// SIMATIC STEP 7 (V5.x) project e009v440
// CPU: CPU 313C-2 DP
// station: P_ADR_BUS
// station: Hardware
// station: PLC Roll Forming
// program: Programa S7(8)
// program: CU320
// program: CU320-2 DP
// program: M440
// program: M440
// program: M440

SYMBOL_TABLE
"Tendencia"	DB 1	DB 1
"EncóderPerfilador"	DB 2	DB 2
"Datos Pieza - Receta"	DB 3	DB 3
"Datos Pieza - Alm1"	DB 4	DB 4
"Datos Pieza - Alm2"	DB 5	DB 5
"Datos Pieza - Araña"	DB 6	DB 6
"Datos Pieza - Rolos"	DB 7	DB 7
"Datos Pieza - Perfilador"	DB 8	DB 8
"Datos Pieza - Cinta"	DB 9	DB 9
"Datos Pieza - Pinza"	DB 10	DB 10
"Datos Pieza - Plegadores"	DB 11	DB 11
"Datos Pieza - Descargado"	DB 12	DB 12
"Posiciones_Pinza"	DB 13	DB 13
"Datos Pieza - VACIO"	DB 14	DB 14
"Ultimo Estado"	DB 15	DB 15
"Datos Cosntructivos"	DB 16	DB 16
"Posiciones Pinza 00"	DB 17	DB 17
"Posiciones_Pinza_Ant"	DB 18	DB 18
"DB Asistencia"	DB 19	DB 19
"ReglasBalluff"	DB 20	DB 20
"Referenciado"	DB 21	DB 21
"Posiciones_Pinza_Ant2"	DB 23	DB 23
"Posiciones_Pinza_Ant3"	DB 24	DB 24
"PosReal_Pinza"	DB 25	DB 25
"PosReal_Pinza_Ant"	DB 26	DB 26
"PosReal_Pinza_Ant2"	DB 27	DB 27
"PosReal_Pinza_Ant3"	DB 28	DB 28
"Error_Pinza_Ant"	DB 29	DB 29
"DB_OP"	DB 50	DB 50
"Recetas"	DB 51	DB 51
"OFFSET"	DB 52	DB 52
"Posiciones Pinza"	DB 53	DB 53
"Posiciones Plegador 2"	DB 54	DB 54
"Posiciones Plegador 1"	DB 55	DB 55
"Posiciones Plegadores 00"	DB 56	DB 56
"Posiciones Pleg. 1 Ant"	DB 57	DB 57
"Posiciones Pleg. 2 Ant"	DB 58	DB 58
"Homing Plegadores"	FC 1	FC 1
"ModoMix"	FC 2	FC 2
"Manual Selección Mov."	FC 4	FC 4
"General"	FC 5	FC 5
"Generador de Fallas"	FC 6	FC 6
"Asistencia"	FC 8	FC 8
"Control de Plegadora"	FC 9	FC 9
"Perfilador"	FC 10	FC 10
"Transportes"	FC 11	FC 11
"Control de Pinza y Forma"	FC 12	FC 12
"Controlador Posiciones"	FC 13	FC 13
"Almacenes"	FC 15	FC 15
"Registro_pos_Plegador"	FC 17	FC 17
"Registro_pos_Pinza"	FC 18	FC 18
"Araña"	FC 20	FC 20
"Plegadora"	FC 30	FC 30
"Plegador 1"	FC 31	FC 31
"Descarga"	FC 40	FC 40
"TR_MP"	FC 50	FC 50
"Gestión de Datos"	FC 51	FC 51
"eProC - Máquina Estados"	FC 150	FC 150
"23S1"	I 0.0	BOOL	// Pupitre Almacenes - Rearme
"23SH2"	I 0.1	BOOL	// Pupitre Almacenes - Reconocimiento
"Pair"	I 0.2	BOOL	// Presión de Aire
"GH_Tmax"	I 0.3	BOOL	// Grupo áulico (23S8) - Temperatura máxima
"23S3"	I 0.4	BOOL	// Pupitre Principal : Rearme
"23S5"	I 0.5	BOOL	// Alineador Eje Y Plegador 1 ON
"23S6"	I 0.6	BOOL	// Alineador Eje Y Plegador 1 OFF
"23S4"	I 0.7	BOOL	// Presostato Freno Perfilador
"24S1_01"	I 1.0	BOOL	// Rueda Unidades :1
"24S1_02"	I 1.1	BOOL	// Rueda Unidades :2
"24S1_04"	I 1.2	BOOL	// Rueda Unidades :4
"24S1_08"	I 1.3	BOOL	// Rueda Unidades :8
"24S1_10"	I 1.4	BOOL	// Rueda Decenas :1
"24S1_20"	I 1.5	BOOL	// Rueda Decenas :2
"24S1_40"	I 1.6	BOOL	// Rueda Decenas :4
"24S1_80"	I 1.7	BOOL	// Rueda Decenas :8
"QF9"	I 2.0	BOOL	// Térmico Freno Ajuste de Formado
"25S2"	I 2.1	BOOL	// Desaceleración Transporte Cinta
"25S3"	I 2.2	BOOL	// Fin de Carrera Araña Arriba
"25S4"	I 2.3	BOOL	// Pistón 1 Araña Contraído
"25S5"	I 2.4	BOOL	// Fin de Carrera Araña Abajo
"25S6"	I 2.5	BOOL	// Araña Abajo
"25S7"	I 2.6	BOOL	// Pistón 2 Araña Expandido
"25S8"	I 2.7	BOOL	// Pistón 2 Araña Contraído
"26S1"	I 3.0	BOOL	// Tulipas no apoyadas en Chapa
"26S2"	I 3.1	BOOL	// Araña en Posicion de Carga
"26S3"	I 3.2	BOOL	// Araña en Posición de Descarga
"26S4"	I 3.3	BOOL	// Bajar Velocidad Transporte de Araña para Tomar Chapa
"26S5"	I 3.4	BOOL	// Bajar Velocidad Transporte de Araña para Soltar Chapa
"26S6"	I 3.5	BOOL	// Presencia de Almacén 2 en Puesto de Espera
"26S7"	I 3.6	BOOL	// Presencia de Almacén 2 en Puesto de Trabajo
"26S8"	I 3.7	BOOL	// Presencia de Chapa en Transporte Rolos
"27S1"	I 4.0	BOOL	// Pulsador Avance Perfilador
"27S2"	I 4.1	BOOL	// Pulsador Retroceso Perfilador
"27S3"	I 4.2	BOOL	// Chapa en entrada Perfilador
"27S4"	I 4.3	BOOL	// Chapa en salida Perfilador
"27S5"	I 4.4	BOOL	// Formador Herramienta 1 Martillo Off
"27S6"	I 4.5	BOOL	// Formador Herramienta 1 Martillo On
"27S7"	I 4.6	BOOL	// Formador Herramienta 1 Matriz Off
"27S8"	I 4.7	BOOL	// Formador Herramienta 1 Matriz On
"28S1"	I 5.0	BOOL	// Formador Herramienta 2 Martillo Off
"28S2"	I 5.1	BOOL	// Formador Herramienta 2 Martillo On
"28S3"	I 5.2	BOOL	// Formador Herramienta 2 Matriz Off
"28S4"	I 5.3	BOOL	// Formador Herramienta 2 Matriz On
"28S5"	I 5.4	BOOL	// Formador Bloqueo Herramienta On
"28S6"	I 5.5	BOOL	// Matriz Formadora Bloqueo Herramienta Off
"28S7"	I 5.6	BOOL	// Ajuste Formador Fin de Carrera Mín.
"28S8"	I 5.7	BOOL	// Ajuste Formador Fin de Carrera Máx.
"29S1"	I 6.0	BOOL	// Formador Bloqueo de avance On
"29S2"	I 6.1	BOOL	// Formador Bloqueo de avance Off
"29S3"	I 6.2	BOOL	// Presencia de Chapa en Formador
"29S4"	I 6.3	BOOL	// Pinza Abierta
"29S5"	I 6.4	BOOL	// Pinza Cerrada
"29S6"	I 6.5	BOOL	// Ajuste Ancho Perfilador Fin de carrera Mín.
"29S7"	I 6.6	BOOL	// Ajuste Ancho Perfilador Fin de carrera Máx.
"29S8"	I 6.7	BOOL	// Plegadora Termostato Grupo Hidráulico
"30S1"	I 7.0	BOOL	// Plegadora Tenaza adelante
"30S2"	I 7.1	BOOL	// Plegadora Tenaza atrás
"30S3"	I 7.2	BOOL	// Plegadora Tenaza arriba
"30S4"	I 7.3	BOOL	// Plegadora Tenaza abajo
"30S5"	I 7.4	BOOL	// Plegadora Tenaza abierta
"30S6"	I 7.5	BOOL	// Plegadora Tenaza cerrada
"30S7"	I 7.6	BOOL	// Plegador 1 Cepillos Arriba
"30S8"	I 7.7	BOOL	// Plegador 1 Cepillos Abajo
"31S1"	I 8.0	BOOL	// Presencia de Producto en Descargador
"31S2"	I 8.1	BOOL	// Descargador Adelante
"31S3"	I 8.2	BOOL	// Descargador Atrás
"31S4"	I 8.3	BOOL	// Barrera Seguridad Descargador
"31S5"	I 8.4	BOOL	// Plegador 1 Fijación Arriba
"31S6"	I 8.5	BOOL	// Plegador 1 Fijación Abajo
"31S7"	I 8.6	BOOL	// Plegador 1 Arriba
"31S8"	I 8.7	BOOL	// Pieza en Descargador
"32S1"	I 9.0	BOOL	// Plegador 1 Prensa Abajo
"32S2"	I 9.1	BOOL	// Plegador 1 Prensa Arriba
"32S3"	I 9.2	BOOL	// Plegador 1 Extensión 1 Prensa Abajo
"32S4"	I 9.3	BOOL	// Plegador 1 Extensión 1 Prensa Arriba
"32S5"	I 9.4	BOOL	// Plegador 1 Extensión 2 Prensa Abajo
"32S6"	I 9.5	BOOL	// Plegador 1 Extensión 2 Prensa Arriba
"QM13.2"	I 9.6	BOOL	// Térmico Refrigeración Grupo Hidráulico Plegadora
"QM14"	I 9.7	BOOL	// Térmico Calentador de Chapa
"QM01"	I 10.0	BOOL	// Térmico Intercambiador de Almacenes
"VAR02"	I 10.1	BOOL	// Defecto Variador Araña
"VAR03"	I 10.2	BOOL	// Defecto Variador Transporte Rolos
"Reserva"	I 10.3	BOOL	// Reserva
"Reserva2"	I 10.4	BOOL	// Reserva
"Doble_Chapa_Perf"	I 10.5	BOOL	// Doble Espesor de Chapa en entrada de Perfilador
"Reserva3"	I 10.6	BOOL	// Reserva
"QM05"	I 10.7	BOOL	// Térmico Bombas de Lubricación Perfilador
"QM06"	I 11.0	BOOL	// Térmico Grupo Hidráulico Freno Perfilador
"QM07"	I 11.1	BOOL	// Térmico Ajuste de Ancho Perfilador
"VAR08"	I 11.2	BOOL	// Defecto Variador Transporte Cinta
"QM09"	I 11.3	BOOL	// Térmico Ajuste de Formado
"Sinamics_OK"	I 11.4	BOOL	// Smart Line Plegador Listo
"Sinamics_Alarme"	I 11.5	BOOL	// Defecto SmartLine Plegadora
"Carter"	I 11.6	BOOL	// Cubierta Perfilador abierta
"QM13.1"	I 11.7	BOOL	// Térmico Grupo Hidráulico Plegadora
"35S1"	I 12.0	BOOL	// Plegador 2 Fijación Arriba
"35S2"	I 12.1	BOOL	// Plegador 2 Fijación Abajo
"35S3"	I 12.2	BOOL	// Plegador 2 Arriba
"35S4"	I 12.3	BOOL	// Plegador 2 Abajo
"35S5"	I 12.4	BOOL	// Plegador 2 Prensa Abajo
"35S6"	I 12.5	BOOL	// Plegador 2 Prensa Arriba
"35S7"	I 12.6	BOOL	// Plegador 2 Extensión 1 Prensa Abajo
"35S8"	I 12.7	BOOL	// Plegador 2 Extensión 1 Prensa Arriba
"36S7"	I 13.0	BOOL	// Plegador 2 Extensión 2 Prensa Abajo
"36S8"	I 13.1	BOOL	// Plegador 2 Extensión 2 Prensa Arriba
"36S1"	I 13.2	BOOL	// Alineador Eje X Plegador 2 ON
"36S2"	I 13.3	BOOL	// Alineador Eje X Plegador 2 OFF
"36S3"	I 13.4	BOOL	// Alineador Eje Y Plegador 2 ON
"36S4"	I 13.5	BOOL	// Alineador Eje Y Plegador 2 OFF
"36S5"	I 13.6	BOOL	// Plegador 2 Cepillos Arriba
"36S6"	I 13.7	BOOL	// Plegador 2 Cepillos Abajo
"36S9"	I 14.0	BOOL	// Plegador 1 Prensa en Posición Intermedia
"36S17"	I 14.1	BOOL	// Plegador 2 Prensa en Posición Intermedia
"36S11"	I 14.2	BOOL	// Pinza Plegadora en Posición Intermedia
"36S12"	I 14.3	BOOL	// Descargador en Posición Intermedia
"36S13"	I 14.4	BOOL	// Atasco Perfilador Sensor 1
"36S14"	I 14.5	BOOL	// Atasco Perfilador Sensor 2
"36S15"	I 14.6	BOOL	// Atasco Perfilador Sensor 3
"36S16"	I 14.7	BOOL	// Atasco Perfilador Sensor 4
"36S10"	I 15.0	BOOL	// Barrera Almacenes
"36S18"	I 15.1	BOOL
"Reserva4"	I 15.2	BOOL	// Reserva
"iPLs_HabAlmacenes"	I 15.3	BOOL	// Pulsador Habilitación Almacenes
"iSel_Homming"	I 15.4	BOOL	// Selectora Habilitación Referenciado Plegadores
"31S7b"	I 15.5	BOOL	// Plegador 1 posición Arriba (pata)
"35S3b"	I 15.6	BOOL	// Plegador 2 posición Arriba (pata)
"36S70"	I 15.7	BOOL	// Barrera Atasco en Perfilador
"Atasco_6"	I 16.0	BOOL	// Sensor 6 Atasco Perfilador
"Atasco_7"	I 16.1	BOOL	// Sensor 7 Atasco Perfilador
"Atasco_8"	I 16.2	BOOL	// Sensor 8 Atasco Perfilador
"Atasco_9"	I 16.3	BOOL	// Sensor 9 Atasco Perfilador
"Atasco_10"	I 16.4	BOOL	// Sensor 10 Atasco Perfilador
"Atasco_11"	I 16.5	BOOL	// Sensor 11 Atasco Perfilador
"Atasco_12"	I 16.6	BOOL	// Sensor 12 Atasco Perfilador
"Atasco_13"	I 16.7	BOOL	// Sensor 13 Atasco Perfilador
"Atasco_14"	I 17.0	BOOL	// Sensor 14 Atasco Perfilador
"Atasco_15"	I 17.1	BOOL	// Sensor 15 Atasco Perfilador
"Atasco_16"	I 17.2	BOOL	// Sensor 16 Atasco Perfilador
"Atasco_17"	I 17.3	BOOL	// Sensor 17 Atasco Perfilador
"Atasco_18"	I 17.4	BOOL	// Sensor 18 Atasco Perfilador
"Atasco_19"	I 17.5	BOOL	// Sensor 19 Atasco Perfilador
"Atasco_21"	I 17.6	BOOL	// Sensor 21 Atasco Perfilador
"iSns_Perf_Atasco_16"	I 17.7	BOOL	// Sensor 20 Atasco Perfilador
"Atasco_22"	I 18.0	BOOL	// Sensor 22 Atasco Perfilador
"Atasco_23"	I 18.1	BOOL	// Sensor 23 Atasco Perfilador
"Atasco_24"	I 18.2	BOOL	// Sensor 24 Atasco Perfilador
"Atasco_5"	I 18.3	BOOL	// Sensor 5 Atasco Perfilador
"Safety_Barrera_Entrada"	I 19.0	BOOL	// Entrada desde PLC Safety en reemplazo de barrera de entrada original
"Safety_Corte_1"	I 19.1	BOOL	// Entrada desde PLC Safety para corte 1
"Safety_Corte_2"	I 19.2	BOOL	// Entrada desde PLC Safety para corte 2
"PRF_SLM_DATA0"	I 24.0	BOOL
"PRF_SLM_MS"	I 24.1	BOOL	// SmartLine Perfilador Mando Solicitado
"PRF_SLM_DATA01"	I 24.2	BOOL
"PRF_SLM_PREC"	I 24.3	BOOL	// SmartLine Perfilador Precarga Terminada
"PRF_SLM_CTC"	I 24.4	BOOL	// SmartLine Perfilador Contactor de Red Cerrado
"PRF_SLM_DATA02"	I 24.5	BOOL
"PRF_SLM_DATA03"	I 24.6	BOOL
"PRF_SLM_DATA04"	I 24.7	BOOL
"PRF_SLM_LC"	I 25.0	BOOL	// SmartLine Perfilador Listo Conexión
"PRF_SLM_LS"	I 25.1	BOOL	// SmartLine Perfilador Listo para Servicio
"PRF_SLM_SH"	I 25.2	BOOL	// SmartLine Perfilador Servicio Habilitado
"PRF_SLM_FA"	I 25.3	BOOL	// SmartLine Perfilador Fallo Activo  (0=NO, 1=SI)
"PRF_SLM_DES2A"	I 25.4	BOOL	// SmartLine Perfilador Sin Parada Natural Activa
"PRF_SLM_DES3A"	I 25.5	BOOL	// SmartLine Perfilador Sin Parada Rápida Activa
"PRF_SLM_BC"	I 25.6	BOOL	// SmartLine Perfilador Bloqueo de Conexión Activo
"PRF_SLM_AL"	I 25.7	BOOL	// SmartLine Perfilador Alarma Activa
"PRF_AlarmaActiva"	I 26.1	BOOL	// Alarma activa en CU Perfiladores (1=NO, 0=SI)
"PRF_FalloActivo"	I 26.2	BOOL	// Fallo activo en CU Perfiladores (1=NO, 0=SI)
"PRF_TS"	I 28.0	BOOL	// Perfiladores Tiempo sist. Sincronizado
"PRF_ALP"	I 28.1	BOOL	// Perfiladores Alarma Presente
"PRF_DFP"	I 28.2	BOOL	// Perfiladores Falla Presente
"PRF_AVS"	I 28.3	BOOL	// Perfiladores Aviso de Seguridad Presente
"PRF_DATA07"	I 28.4	BOOL
"PRF_DATA08"	I 28.5	BOOL
"PRF_DATA09"	I 28.6	BOOL
"PRF_DATA10"	I 28.7	BOOL
"PRF_DATA0"	I 29.0	BOOL
"PRF_DATA01"	I 29.1	BOOL
"PRF_DATA03"	I 29.2	BOOL
"PRF_DF"	I 29.3	BOOL	// Perfiladores Fallo Activo
"PRF_DATA04"	I 29.4	BOOL
"PRF_DATA05"	I 29.5	BOOL
"PRF_DATA06"	I 29.6	BOOL
"PRF_AL"	I 29.7	BOOL	// Perfiladores Alarma Activa
"PL1_ecart"	I 62.0	BOOL	// Plegador 1 Error de Seguimiento dentro de Tolerancia
"PL1_PL1lote"	I 62.1	BOOL	// Plegador 1 Mando Solicitado
"PL1_target"	I 62.2	BOOL	// Plegador 1 Posición de destino Alcanzada
"PL1_enreference"	I 62.3	BOOL	// Plegador 1 Punto de Referencia Seteado
"PL1_acquite"	I 62.4	BOOL	// Plegador 1 Confirmación Bloque de Desplazamiento Activada
"PL1_Stopped"	I 62.5	BOOL	// Plegador 1 Detenido
"PL1_Hom1"	I 62.6	BOOL	// Plegador 1 Sensor homing
"DI8_CU_PL"	I 62.7	BOOL	// Límite Plegador 1
"PL1_enclanche"	I 63.0	BOOL	// Plegador 1 Listo Conexión
"PL1_prêt"	I 63.1	BOOL	// Plegador 1 Listo para Servicio
"PL1_fonction"	I 63.2	BOOL	// Plegador 1 Servicio Habilitado
"PL1_defaut"	I 63.3	BOOL	// Plegador 1 Fallo Activo
"PL1_arret2on"	I 63.4	BOOL	// Plegador 1 Sin Parada Natural Activa
"PL1_arret3on"	I 63.5	BOOL	// Plegador 1 Sin Parada Rápida Activa
"PL1_convbloc"	I 63.6	BOOL	// Plegador 1 Bloqueo de Conexión Activo
"PL1_alarme"	I 63.7	BOOL	// Plegador 1 Alarma Activa
"PL1_ReqRR"	I 67.4	BOOL	// Plegador 1 Requiere RAM en ROM
"PL2_ecart"	I 82.0	BOOL	// Plegador 2 Error de Seguimiento dentro de Tolerancia
"PL2_PL2lote"	I 82.1	BOOL	// Plegador 2 Mando Solicitado
"PL2_target"	I 82.2	BOOL	// Plegador 2 Posición de destino Alcanzada
"PL2_enreference"	I 82.3	BOOL	// Plegador 2 Punto de Referencia Seteado
"PL2_acquite"	I 82.4	BOOL	// Plegador 2 Confirmación Bloque de Desplazamiento Activada
"PL2_Stopped"	I 82.5	BOOL	// Plegador 2 Detenido
"PL2_Hom2"	I 82.6	BOOL	// Plegador 2 Sensor Homing
"DI9_CU_PL"	I 82.7	BOOL	// Límite Plegador 2
"PL2_enclanche"	I 83.0	BOOL	// Plegador 2 Listo Conexión
"PL2_prêt"	I 83.1	BOOL	// Plegador 2 Listo para Servicio
"PL2_fonction"	I 83.2	BOOL	// Plegador 2 Servicio Habilitado
"PL2_defaut"	I 83.3	BOOL	// Plegador 2 Fallo Activo
"PL2_arret2on"	I 83.4	BOOL	// Plegador 2 Sin Parada Natural Activa
"PL2_arret3on"	I 83.5	BOOL	// Plegador 2 Sin Parada Rápida Activa
"PL2_convbloc"	I 83.6	BOOL	// Plegador 2 Bloqueo de Conexión Activo
"PL2_alarme"	I 83.7	BOOL	// Plegador 2 Alarma Activa
"PL2_ReqRR"	I 87.4	BOOL	// Plegador 2 Requiere RAM en ROM
"PI_ecart"	I 102.0	BOOL	// Pinza Error de Seguimiento dentro de Tolerancia
"PI_pilote"	I 102.1	BOOL	// Pinza Mando Solicitado
"PI_target"	I 102.2	BOOL	// Pinza Posición de destino Alcanzada
"PI_enreference"	I 102.3	BOOL	// Pinza Punto de Referencia Seteado
"PI_acquite"	I 102.4	BOOL	// Pinza Confirmación Bloque de Desplazamiento Activada
"PI_Stopped"	I 102.5	BOOL	// Pinza Detenida
"CU_Falla"	I 102.6	BOOL	// Cu Plegadora - Falla Presente
"CU_FallaSafety"	I 102.7	BOOL	// Cu Plegadora - Falla Safety Presente
"PI_enclanche"	I 103.0	BOOL	// Pinza Listo Conexión
"PI_prêt"	I 103.1	BOOL	// Pinza Listo para Servicio
"PI_fonction"	I 103.2	BOOL	// Pinza Servicio Habilitado
"PI_defaut"	I 103.3	BOOL	// Pinza Fallo Activo
"PI_arret2on"	I 103.4	BOOL	// Pinza Sin Parada Natural Activa
"PI_arret3on"	I 103.5	BOOL	// Pinza Sin Parada Rápida Activa
"PI_convbloc"	I 103.6	BOOL	// Pinza Bloqueo de Conexión Activo
"PI_alarme"	I 103.7	BOOL	// Pinza Alarma Activa
"KMST"	I 124.0	BOOL	// Baja Tensión
"KMES"	I 124.1	BOOL	// En Servicio
"21SH1"	I 124.2	BOOL	// Parada de Ciclo
"21S2"	I 124.3	BOOL	// Pausar Ciclo
"21S3"	I 124.4	BOOL	// AUTO
"21S4"	I 124.5	BOOL	// Rearme
"21S5"	I 124.6	BOOL	// Alineador Eje X Plegador 1 ON
"21S6"	I 124.7	BOOL	// Alineador Eje X Plegador 1 OFF
"22S1_01"	I 125.0	BOOL	// Rueda Unidades :1
"22S1_02"	I 125.1	BOOL	// Rueda Unidades :2
"22S1_04"	I 125.2	BOOL	// Rueda Unidades :4
"22S1_08"	I 125.3	BOOL	// Rueda Unidades :8
"22S1_10"	I 125.4	BOOL	// Rueda Decenas :1
"22S1_20"	I 125.5	BOOL	// Rueda Decenas :2
"22S1_40"	I 125.6	BOOL	// Rueda Decenas :4
"22S1_80"	I 125.7	BOOL	// Rueda Decenas :8
"DF_Perlfilador1"	I 257.0	BOOL	// Defecto en Motor Perfilador 1
"DF_Perlfilador2"	I 257.1	BOOL	// Defecto en Motor Perfilador 2
"DF_Perlfilador3"	I 257.2	BOOL	// Defecto en Motor Perfilador 3
"DF_Perlfilador4"	I 257.3	BOOL	// Defecto en Motor Perfilador 4
"DF_CU_PERFI"	I 259.0	BOOL	// Fallo en Cu Perfiladora
"CU_FinRAM_ROM"	I 259.2	BOOL	// CU finaliza la carga de RAM en ROM
"COD1_VALEUR"	ID 40	DINT	// Encóder Perfilador
"COD2_VALEUR"	ID 44	DINT	// Encoder Formador
"PL1_cote"	ID 72	DINT	// Plegador 1 Posición Actual
"PL2_cote"	ID 92	DINT	// Plegador 2 Posición Actual
"PI_cote"	ID 112	DINT	// Pinza Posición Actual
"VAR_02_Etat"	IW 50	INT	// Variador Araña Status Word
"VAR_02_RVitesse"	IW 52	INT	// Variador Araña Velocidad Real
"VAR_03_Etat"	IW 54	INT	// Variador Rolos Araña Status Word
"VAR_03_RVitesse"	IW 56	INT	// Variador Rolos Araña Velocidad Real
"VAR_08_Etat"	IW 58	INT	// Variador Cinta Transporte Status Word
"VAR_08_RVitesse"	IW 60	INT	// Variador Cinta Transporte Velocidad Real
"Bit 0"	M 0.0	BOOL	// Bit en 0
"Bit 1"	M 0.1	BOOL	// Bit en 1
"PRF_BRR_SDF"	M 0.4	BOOL	// Barrera Perfilador Sin Atasco
"Ar_Enc"	M 0.5	BOOL	// Enclavamiento Araña
"ACQUIT"	M 0.6	BOOL	// Reconocer Defecto
"Hab_PLC_Plegadores"	M 0.7	BOOL	// Habilitación de Plegadores desde el PLC
"DCH_GH_cmd"	M 1.0	BOOL	// Descargador : Requerimiento de marcha Grupo áulico
"PL1_GH_cmd"	M 1.1	BOOL	// Plegador 1 : Requerimiento de marcha Grupo Hidráulico
"PL2_GH_cmd"	M 1.2	BOOL	// Plegador 2 : Requerimiento de marcha Grupo Hidráulico
"FO_GH_cmd"	M 1.3	BOOL	// Formador : Requerimiento de marcha Grupo áulico
"GH_verrou"	M 1.5	BOOL	// Enclavamiento Grupo áulico
"REF_OPT"	M 2.0	BOOL	// Refrigeración Grupo Hidráulico
"Ant_Fijacion1"	M 4.0	BOOL	// Anticipación Fijación Plegador 1
"Ant_Fijacion2"	M 4.1	BOOL	// Anticipación Fijación Plegador 2
"AnT_Desc"	M 4.7	BOOL	// Antiscipar descargador
"VAR_PERF_OK"	M 6.0	BOOL	// Variador Perfilador en Falla
"DRIVES_PERF_OK"	M 6.1	BOOL	// Drives Perfilador en Falla
"Clk_0.1s"	M 9.0	BOOL
"Clk_0.2s"	M 9.1	BOOL
"Clk_0.4s"	M 9.2	BOOL
"Clk_0.5s"	M 9.3	BOOL
"Clk_0.8s"	M 9.4	BOOL
"Clk_1s"	M 9.5	BOOL
"Clk_1.6s"	M 9.6	BOOL
"Clk_2s"	M 9.7	BOOL
"MES"	M 10.0	BOOL	// Puesta en Marcha
"AUTO"	M 10.1	BOOL	// Modo Automático
"MANU"	M 10.2	BOOL	// Modo Manual
"CYCLE"	M 10.3	BOOL	// En Ciclo
"D_FCYC"	M 10.4	BOOL	// Solicitud Fin de Ciclo
"FCYC"	M 10.5	BOOL	// Posición Final de Ciclo
"SAR"	M 10.6	BOOL	// Seguridad Máquinas
"T_ALM2"	M 11.0	BOOL	// Trabajar con  Almacén 2
"T_ALM1"	M 11.1	BOOL	// Trabajar con Almacén 1
"MM1_CONTADOR_FIN"	M 11.2	BOOL	// Contador de Almacén 1 Finalizado
"MM2_CONTADOR_FIN"	M 11.3	BOOL	// Contador de Almacén 2 Finalizado
"AUX_FP_Reset"	M 15.0	BOOL	// Aux flanco positivo orden de Reset
"CA_KM09.1"	M 16.0	BOOL	// Avance Formador
"CA_42K3"	M 16.1	BOOL	// Herramienta 1 Accionar Martillo
"CA_42K5"	M 16.2	BOOL	// Herramienta 1 Accionar Matriz
"CA_42K7"	M 16.3	BOOL	// Herramienta 2 Accionar Martillo
"CA_43K1"	M 16.4	BOOL	// Herramienta 2 Accionar Matriz
"CA_43K3"	M 16.5	BOOL	// Bloqueo de Herramienta Bajar
"CA_43Y5"	M 16.6	BOOL	// Bajar Formador
"CA_43Y7"	M 16.7	BOOL	// Órden Abrir Pinza
"CA_KM09.2"	M 17.0	BOOL	// Retroceso Formador
"F_H_Bloqueadas"	M 17.1	BOOL	// Seguridad Herramientas Bloqueadas
"F_H_Desactivadas"	M 17.2	BOOL	// Seguridad Herramientas Desactivadas
"CA_42K8"	M 17.3	BOOL	// Herramienta 2 Liberar Martillo
"CA_43K2"	M 17.4	BOOL	// Herramienta 2 Liberar Matriz
"CA_43K4"	M 17.5	BOOL	// Liberar Bloqueo de Herramientas
"CA_43Y6"	M 17.6	BOOL	// Formador Subir
"CA_43Y8"	M 17.7	BOOL	// Órden Cerrar Pinza
"CA_KM02_1"	M 18.0	BOOL	// Transporte de Araña Avance Automático
"CA_40Y7"	M 18.1	BOOL	// Araña Subir Pistón Inferior Automático
"CA_41Y2"	M 18.2	BOOL	// Bajar Pistón Superior Automático
"CA_45K1"	M 18.3	BOOL	// Descargador Avance Automático
"CA_KM01_1"	M 18.4	BOOL	// Intercambiador Almacenes Avance (Alm1)
"PH_AV"	M 18.7	BOOL	// Araña en Posición Fuera de Rango
"CA_KM02_2"	M 19.0	BOOL	// Transporte de Araña Retroceso Automático
"CA_41Y1"	M 19.1	BOOL	// Araña Bajar Pistón Inferior Automático
"CA_41Y3"	M 19.2	BOOL	// Subir Pistón Superior Automático
"CA_45K2"	M 19.3	BOOL	// Descargador Retroceso Automático
"CA_KM01_2"	M 19.4	BOOL	// Intercambiador Almacenes Retroceso (Alm2)
"CA_KM04_5"	M 20.0	BOOL	// Perfilador Avance Automático
"CA_44Y3"	M 20.3	BOOL	// Tenaza Plegadora Bajar Automático
"CA_46K5"	M 20.5	BOOL	// PLIEUSES :  condition Auto Taquage X
"CA_46K6"	M 20.6	BOOL	// PLIEUSES :  condition Auto Taquage Y
"CA_46K7"	M 20.7	BOOL	// Plegadora Subir Cepillos Automático
"ANT_RESC"	M 21.1	BOOL	// ESCAMOTEUR : anticipation recul
"FP_46K5"	M 21.5	BOOL	// Plegadora Flanco positivo Alineación X
"FP_46K6"	M 21.6	BOOL	// Plegadora Flanco positivo Alineación Y
"FM_46K7"	M 21.7	BOOL	// Plegadora Orden de Subir Cepillos
"CA_45K3"	M 22.0	BOOL	// Plegador 1 Avance Fijación
"CA_45K5"	M 22.1	BOOL	// Plegador 1 Subir
"CA_45K7"	M 22.2	BOOL	// Plegador 1 V1 Accionar
"CA_46K1"	M 22.3	BOOL	// Plegador 1 V2 Accionar
"CA_47K1"	M 22.4	BOOL	// Plegador 2 Avance Fijación
"CA_47K3"	M 22.5	BOOL	// Plegador 2 Subir
"CA_47K5"	M 22.6	BOOL	// Plegador 2 V1 Accionar
"CA_47K7"	M 22.7	BOOL	// Plegador 2 V2 Accionar
"CA_45K4"	M 23.0	BOOL	// Plegador 1 Retroceso Fijación
"CA_45K6"	M 23.1	BOOL	// Plegador 1 Bajar
"CA_45K8"	M 23.2	BOOL	// Plegador 1 V1 Liberar
"CA_46K2"	M 23.3	BOOL	// Plegador 1 V2 Liberar
"CA_47K2"	M 23.4	BOOL	// Plegador 2 Retroceso Fijación
"CA_47K4"	M 23.5	BOOL	// Plegador 2 Bajar
"CA_47K6"	M 23.6	BOOL	// Plegador 2 V1 Liberar
"CA_47K8"	M 23.7	BOOL	// Plegador 2 V2 Liberar
"CA_46K3"	M 24.0	BOOL	// Plegador 1 V3 Accionar
"CA_46K4"	M 24.1	BOOL	// Plegador 1 V3 Liberar
"CA_48K1"	M 24.2	BOOL	// Plegador 2 V3 Accionar
"CA_48K2"	M 24.3	BOOL	// Plegador 2 V3 Liberar
"PL1_V_PT"	M 24.4	BOOL	// Plegador 1  V1-2-3 Trabajando
"PL2_V_PT"	M 24.5	BOOL	// Plegador 2  V1-2-3 Trabajando
"CA_PI_AV"	M 25.0	BOOL	// Avanzar Pinza
"CA_PI_RC"	M 25.1	BOOL	// Retroceder Pinza
"CA_PI_Target"	M 25.2	BOOL	// Pinza en Posición
"PL_Tenaza_Anticipada"	M 25.3	BOOL	// Tenaza en anticipation
"FOR_COND_H1"	M 26.0	BOOL	// Habilitación Herramienta 1
"FOR_COND_H2"	M 26.1	BOOL	// Habilitación Herramienta 2
"FN_46K5"	M 26.2	BOOL	// Plegadora Flanco negativo Alineación X
"FN_46K6"	M 26.3	BOOL	// Plegadora Flanco negativo Alineación Y
"PI_XP"	M 26.4	BOOL
"FP_46K7"	M 26.5	BOOL	// Plegadora Flanco positivo Subir Cepillos
"FN_46K7"	M 26.6	BOOL	// Plegadora Flanco negativo Subir Cepillos
"CA_PL1_AV"	M 27.0	BOOL	// Plegador 1 Avance
"CA_PL1_RC"	M 27.1	BOOL	// Plegador 1 Retroceso
"CA_PL1_Target"	M 27.2	BOOL	// Plegador 1 en Posición
"CA_PL2_AV"	M 27.4	BOOL	// Plegador 2 Avance
"CA_PL2_RC"	M 27.5	BOOL	// Plegador 2 Retroceso
"CA_PL2_Target"	M 27.6	BOOL	// Plegador 2 en Posición
"PL1_SAR"	M 28.0	BOOL	// Plegador 1 Seguridad
"PL2_SAR"	M 28.4	BOOL	// Plegador 2 Seguridad
"PL_DT"	M 29.0	BOOL	// Solicitud de Plegado
"PL_FT"	M 29.1	BOOL	// Fin de Plegado
"PL_AD"	M 29.2	BOOL	// Plegadora Autorización de desplazamiento
"PL_MT1"	M 29.3	BOOL	// Memoria de Trabajo Plegadora
"PL_V1max"	M 29.4	BOOL	// Plegadora Autorización de desplazamiento Maxi V1
"VAL_RC1"	M 35.0	BOOL	// Validación de movimiento Rueda 1
"VAL_RC2"	M 35.1	BOOL	// Validación de movimiento Rueda 2
"FM_RC1"	M 35.2	BOOL	// Validación de movimiento Rueda 1
"FM_RC2"	M 35.3	BOOL	// Validación de movimiento Rueda 2
"SEL_MANU1"	M 35.6	BOOL	// Selección Manual 1
"SEL_MANU2"	M 35.7	BOOL	// Selección Manual 2
"FM_43Y6"	M 37.6	BOOL	// Formador Arriba
"FM_36S13"	M 40.4	BOOL	// Atasco Perfilador 1
"FM_36S14"	M 40.5	BOOL	// Atasco Perfilador 2
"FM_36S15"	M 40.6	BOOL	// Atasco Perfilador 3
"FM_36S16"	M 40.7	BOOL	// Atasco Perfilador 4
"PRF_HAB_S12"	M 41.0	BOOL	// Perfilador Habilitar detección transición 1-2
"PRF_HAB_S23"	M 41.1	BOOL	// Perfilador Habilitar detección transición 2-3
"PRF_HAB_S34"	M 41.2	BOOL	// Perfilador Habilitar detección transición 3-4
"PRF_HAB_S45"	M 41.3	BOOL	// Perfilador Habilitar detección transición 4-5
"PRF_HAB_S56"	M 41.4	BOOL	// Perfilador Habilitar detección transición 5-6
"PRF_HAB_S67"	M 41.5	BOOL	// Perfilador Habilitar detección transición 6-7
"PRF_HAB_S78"	M 41.6	BOOL	// Perfilador Habilitar detección transición 7-8
"PRF_HAB_S89"	M 41.7	BOOL	// Perfilador Habilitar detección transición 8-9
"PRF_HAB_S910"	M 42.0	BOOL	// Perfilador Habilitar detección transición 9-10
"PRF_HAB_S1011"	M 42.1	BOOL	// Perfilador Habilitar detección transición 10-11
"PRF_HAB_S1112"	M 42.2	BOOL	// Perfilador Habilitar detección transición 11-12
"PRF_HAB_S1213"	M 42.3	BOOL	// Perfilador Habilitar detección transición 12-13
"PRF_HAB_S1314"	M 42.4	BOOL	// Perfilador Habilitar detección transición 13-14
"PRF_HAB_S1415"	M 42.5	BOOL	// Perfilador Habilitar detección transición 14-15
"PRF_HAB_S1516"	M 42.6	BOOL	// Perfilador Habilitar detección transición 15-16
"PRF_HAB_S1617"	M 42.7	BOOL	// Perfilador Habilitar detección transición 16-17
"PRF_HAB_S1718"	M 43.0	BOOL	// Perfilador Habilitar detección transición 17-18
"PRF_HAB_S1819"	M 43.1	BOOL	// Perfilador Habilitar detección transición 18-19
"PRF_HAB_S1920"	M 43.2	BOOL	// Perfilador Habilitar detección transición 19-20
"Simul_conf_Alineadores"	M 62.2	BOOL
"Restart_PLC"	M 62.4	BOOL
"RC1_52"	M 64.0	BOOL	// Rueda RC1 en valor 52
"RC1_53"	M 64.1	BOOL	// Rueda RC1 en valor 53
"RC1_54"	M 64.2	BOOL	// Rueda RC1 en valor 54
"RC1_55"	M 64.3	BOOL	// Rueda RC1 en valor 55
"RC1_56"	M 64.4	BOOL	// Rueda RC1 en valor 56
"RC1_20"	M 66.0	BOOL	// Rueda RC1 en valor 20
"RC1_21"	M 66.1	BOOL	// Rueda RC1 en valor 21
"RC1_22"	M 66.2	BOOL	// Rueda RC1 en valor 22
"RC1_23"	M 66.3	BOOL	// Rueda RC1 en valor 23
"RC1_24"	M 66.4	BOOL	// Rueda RC1 en valor 24
"RC1_25"	M 66.5	BOOL	// Rueda RC1 en valor 25
"RC1_26"	M 66.6	BOOL	// Rueda RC1 en valor 26
"RC1_27"	M 66.7	BOOL	// Rueda RC1 en valor 27
"RC1_28"	M 67.0	BOOL	// Rueda RC1 en valor 28
"RC1_29"	M 67.1	BOOL	// Rueda RC1 en valor 29
"RC1_30"	M 67.2	BOOL	// Rueda RC1 en valor 30
"RC1_31"	M 67.3	BOOL	// Rueda RC1 en valor 31
"RC1_32"	M 67.4	BOOL	// Rueda RC1 en valor 32
"RC1_33"	M 67.5	BOOL	// Rueda RC1 en valor 33
"RC1_34"	M 67.6	BOOL	// Rueda RC1 en valor 34
"RC1_35"	M 67.7	BOOL	// Rueda RC1 en valor 35
"RC1_36"	M 68.0	BOOL	// Rueda RC1 en valor 36
"RC1_37"	M 68.1	BOOL	// Rueda RC1 en valor 37
"RC1_38"	M 68.2	BOOL	// Rueda RC1 en valor 38
"RC1_39"	M 68.3	BOOL	// Rueda RC1 en valor 39
"RC1_40"	M 68.4	BOOL	// Rueda RC1 en valor 40
"RC1_41"	M 68.5	BOOL	// Rueda RC1 en valor 41
"RC1_42"	M 68.6	BOOL	// Rueda RC1 en valor 42
"RC1_43"	M 68.7	BOOL	// Rueda RC1 en valor 43
"RC1_44"	M 69.0	BOOL	// Rueda RC1 en valor 44
"RC1_45"	M 69.1	BOOL	// Rueda RC1 en valor 45
"RC1_46"	M 69.2	BOOL	// Rueda RC1 en valor 46
"RC1_47"	M 69.3	BOOL	// Rueda RC1 en valor 47
"RC1_48"	M 69.4	BOOL	// Rueda RC1 en valor 48
"RC1_49"	M 69.5	BOOL	// Rueda RC1 en valor 49
"RC1_50"	M 69.6	BOOL	// Rueda RC1 en valor 50
"RC1_51"	M 69.7	BOOL	// Rueda RC1 en valor 51
"AuxFn_0"	M 70.0	BOOL
"AuxFn_1"	M 70.1	BOOL
"AuxFn_2"	M 70.2	BOOL
"AuxFn_3"	M 70.3	BOOL
"AuxFn_4"	M 70.4	BOOL
"AuxFn_5"	M 70.5	BOOL
"AuxFn_6"	M 70.6	BOOL
"AuxFn_7"	M 70.7	BOOL
"AuxFn_8"	M 71.0	BOOL
"AuxFn_9"	M 71.1	BOOL
"AuxFn_10"	M 71.2	BOOL
"AuxFn_11"	M 71.3	BOOL
"AuxFn_12"	M 71.4	BOOL
"AuxFn_13"	M 71.5	BOOL
"AuxFn_14"	M 71.6	BOOL
"AuxFn_15"	M 71.7	BOOL
"AuxFn_16"	M 72.0	BOOL
"AuxFn_17"	M 72.1	BOOL
"AuxFn_18"	M 72.2	BOOL
"AuxFn_19"	M 72.3	BOOL
"AuxFn_20"	M 72.4	BOOL
"AuxFn_21"	M 72.5	BOOL
"AuxFn_22"	M 72.6	BOOL
"Reset_Temp_Atasco"	M 72.7	BOOL
"AuxFp_MM1"	M 75.0	BOOL
"AuxFp_MM2"	M 75.1	BOOL
"Desactivar_Falla1"	M 80.0	BOOL
"Desactivar_Falla2"	M 80.1	BOOL
"Desactivar_Falla3"	M 80.2	BOOL
"Desactivar_Falla4"	M 80.3	BOOL
"Desactivar_Falla5"	M 80.4	BOOL
"Desactivar_Falla6"	M 80.5	BOOL
"Desactivar_Falla7"	M 80.6	BOOL
"Desactivar_Falla8"	M 80.7	BOOL
"Desactivar_Falla9"	M 81.0	BOOL
"Desactivar_Falla10"	M 81.1	BOOL
"Desactivar_Falla11"	M 81.2	BOOL
"Desactivar_Falla12"	M 81.3	BOOL
"Desactivar_Falla13"	M 81.4	BOOL
"Desactivar_Falla14"	M 81.5	BOOL
"Desactivar_Falla15"	M 81.6	BOOL
"Desactivar_Falla16"	M 81.7	BOOL
"Desactivar_Falla17"	M 82.0	BOOL
"Desactivar_Falla18"	M 82.1	BOOL
"Desactivar_Falla19"	M 82.2	BOOL
"Desactivar_Falla20"	M 82.3	BOOL
"Desactivar_Falla21"	M 82.4	BOOL
"Desactivar_Falla22"	M 82.5	BOOL
"Desactivar_Falla23"	M 82.6	BOOL
"Desactivar_Falla24"	M 82.7	BOOL
"Desactivar_Falla25"	M 83.0	BOOL
"Desactivar_Falla26"	M 83.1	BOOL
"Desactivar_Falla27"	M 83.2	BOOL
"Desactivar_Falla28"	M 83.3	BOOL
"Desactivar_Falla29"	M 83.4	BOOL
"Desactivar_Falla30"	M 83.5	BOOL
"Desactivar_Falla31"	M 83.6	BOOL
"Desactivar_Falla32"	M 83.7	BOOL
"Desactivar_Falla33"	M 84.0	BOOL
"Desactivar_Falla34"	M 84.1	BOOL
"Desactivar_Falla35"	M 84.2	BOOL
"Desactivar_Falla36"	M 84.3	BOOL
"Desactivar_Falla37"	M 84.4	BOOL
"Desactivar_Falla38"	M 84.5	BOOL
"Desactivar_Falla39"	M 84.6	BOOL
"Desactivar_Falla40"	M 84.7	BOOL
"Desactivar_Falla41"	M 85.0	BOOL
"Desactivar_Falla42"	M 85.1	BOOL
"Desactivar_Falla43"	M 85.2	BOOL
"Desactivar_Falla44"	M 85.3	BOOL
"Desactivar_Falla45"	M 85.4	BOOL
"Desactivar_Falla46"	M 85.5	BOOL
"Desactivar_Falla47"	M 85.6	BOOL
"Desactivar_Falla48"	M 85.7	BOOL
"Desactivar_Falla49"	M 86.0	BOOL
"Desactivar_Falla50"	M 86.1	BOOL
"Desactivar_Falla51"	M 86.2	BOOL
"Desactivar_Falla52"	M 86.3	BOOL
"Desactivar_Falla53"	M 86.4	BOOL
"Desactivar_Falla54"	M 86.5	BOOL
"Desactivar_Falla55"	M 86.6	BOOL
"Desactivar_Falla56"	M 86.7	BOOL
"Desactivar_Falla57"	M 87.0	BOOL
"Desactivar_Falla58"	M 87.1	BOOL
"Desactivar_Falla59"	M 87.2	BOOL
"Desactivar_Falla60"	M 87.3	BOOL
"Desactivar_Falla61"	M 87.4	BOOL
"Desactivar_Falla62"	M 87.5	BOOL
"Desactivar_Falla63"	M 87.6	BOOL
"Desactivar_Falla64"	M 87.7	BOOL
"Desactivar_Falla65"	M 88.0	BOOL
"Desactivar_Falla66"	M 88.1	BOOL
"Desactivar_Falla67"	M 88.2	BOOL
"Desactivar_Falla68"	M 88.3	BOOL
"Desactivar_Falla69"	M 88.4	BOOL
"Desactivar_Falla70"	M 88.5	BOOL
"Desactivar_Falla71"	M 88.6	BOOL
"Desactivar_Falla72"	M 88.7	BOOL
"Desactivar_Falla73"	M 89.0	BOOL
"Desactivar_Falla74"	M 89.1	BOOL
"Desactivar_Falla75"	M 89.2	BOOL
"Desactivar_Falla76"	M 89.3	BOOL
"Desactivar_Falla77"	M 89.4	BOOL
"Desactivar_Falla78"	M 89.5	BOOL
"Desactivar_Falla79"	M 89.6	BOOL
"Desactivar_Falla80"	M 89.7	BOOL
"Desactivar_Falla81"	M 90.0	BOOL
"Desactivar_Falla82"	M 90.1	BOOL
"Desactivar_Falla83"	M 90.2	BOOL
"Desactivar_Falla84"	M 90.3	BOOL
"Desactivar_Falla85"	M 90.4	BOOL
"Desactivar_Falla86"	M 90.5	BOOL
"Desactivar_Falla87"	M 90.6	BOOL
"Desactivar_Falla88"	M 90.7	BOOL
"Desactivar_Falla89"	M 91.0	BOOL
"Desactivar_Falla90"	M 91.1	BOOL
"Desactivar_Falla91"	M 91.2	BOOL
"Desactivar_Falla92"	M 91.3	BOOL
"Desactivar_Falla93"	M 91.4	BOOL
"Desactivar_Falla94"	M 91.5	BOOL
"Desactivar_Falla95"	M 91.6	BOOL
"Desactivar_Falla96"	M 91.7	BOOL
"Desactivar_Falla97"	M 92.0	BOOL
"Desactivar_Falla98"	M 92.1	BOOL
"Desactivar_Falla99"	M 92.2	BOOL
"Desactivar_Falla100"	M 92.3	BOOL
"Desactivar_Falla101"	M 92.4	BOOL
"Desactivar_Falla102"	M 92.5	BOOL
"Desactivar_Falla103"	M 92.6	BOOL
"Desactivar_Falla104"	M 92.7	BOOL
"Desactivar_Falla105"	M 93.0	BOOL
"Desactivar_Falla106"	M 93.1	BOOL
"Desactivar_Falla107"	M 93.2	BOOL
"Desactivar_Falla108"	M 93.3	BOOL
"Desactivar_Falla109"	M 93.4	BOOL
"Desactivar_Falla110"	M 93.5	BOOL
"Desactivar_Falla111"	M 93.6	BOOL
"Desactivar_Falla112"	M 93.7	BOOL
"Desactivar_Falla113"	M 94.0	BOOL
"Desactivar_Falla114"	M 94.1	BOOL
"Desactivar_Falla115"	M 94.2	BOOL
"Desactivar_Falla116"	M 94.3	BOOL
"Desactivar_Falla117"	M 94.4	BOOL
"Desactivar_Falla118"	M 94.5	BOOL
"Desactivar_Falla119"	M 94.6	BOOL
"Desactivar_Falla120"	M 94.7	BOOL
"Desactivar_Falla121"	M 95.0	BOOL
"Desactivar_Falla122"	M 95.1	BOOL
"Desactivar_Falla123"	M 95.2	BOOL
"Desactivar_Falla124"	M 95.3	BOOL
"Desactivar_Falla125"	M 95.4	BOOL
"Alarma_Almacenes"	M 96.0	BOOL
"Alarma_Araña"	M 96.1	BOOL
"Alarma_Rolos"	M 96.2	BOOL
"Alarma_Perfiladores"	M 96.3	BOOL
"Alarma_Cinta"	M 96.4	BOOL
"Alarma_Formador"	M 96.5	BOOL
"Alarma_Pinza"	M 96.6	BOOL
"Alarma_Plegador"	M 96.7	BOOL
"Alarma_Descargador"	M 97.0	BOOL
"Alarma_General"	M 97.1	BOOL
"PL_Req_Pos_Recepción"	M 100.0	BOOL	// Plegadores requieren Posición de Recepción
"PL_Req_Pos_Alineacion"	M 100.1	BOOL	// Plegadores requieren Posición de Alineación
"PL_Req_Pos_Plegado1"	M 100.2	BOOL	// Plegadores requieren Posición de Plegado 1
"PL_Req_Pos_Plegado2"	M 100.3	BOOL	// Plegadores requieren Posición de Plegado 2
"PL_Req_Pos_Entrega"	M 100.4	BOOL	// Plegadores requieren Posición de Entrega
"PL_Req_Pos_Espera"	M 100.5	BOOL	// Plegadores requieren Posición de Espera
"PL_PL1_Posicionando"	M 100.6	BOOL	// Plegador 1 Posicionando
"PL_PL2_Posicionando"	M 100.7	BOOL	// Plegador 2 Posicionando
"Err_P_PL"	M 101.0	BOOL	// Error Prioritarias Máquina de Estados Plegadora
"Err_C_PL"	M 101.1	BOOL	// Error Concatenadoras Máquina de Estados Plegadora
"STOP_RUN"	M 101.3	BOOL	// Cambio de estado Stop a Run
"PL_Rearranque"	M 101.4	BOOL	// Rearranque de máquina de estados
"PL_Continuar"	M 101.5	BOOL	// Continuar con el último estado
"PI_Posicionando"	M 101.6	BOOL	// Posicionando Pinza
"Aux_Clk"	M 102.0	BOOL
"Aux_Pieza_DC"	M 102.1	BOOL
"Aux_Clk2"	M 102.2	BOOL
"Aux_Clk3"	M 102.3	BOOL
"Aux_Clk4"	M 102.4	BOOL
"Aux_Clk5"	M 102.5	BOOL
"Hab_Medición"	M 102.6	BOOL
"Aux_ProD"	M 103.0	BOOL
"Reset_ProD"	M 103.1	BOOL
"PI_Req_Pos_E1H1"	M 104.0	BOOL	// Pinza requiere Posición de Esquina 1 Herramienta 1
"PI_Req_Pos_E1H2"	M 104.1	BOOL	// Pinza requiere Posición de Esquina 1 Herramienta 2
"PI_Req_Pos_E2H1"	M 104.2	BOOL	// Pinza requiere Posición de Esquina 2 Herramienta 1
"PI_Req_Pos_E2H2"	M 104.3	BOOL	// Pinza requiere Posición de Esquina 2 Herramienta 2
"PI_Req_Pos_Entrega"	M 104.4	BOOL	// Pinza requiere Posición de Entrega
"PI_Req_Pos_Inicial"	M 104.5	BOOL	// Pinza requiere Posición de Recepción
"Warning 1"	M 110.0	BOOL
"Warning 2"	M 110.1	BOOL
"Warning 3"	M 110.2	BOOL
"Warning 4"	M 110.3	BOOL
"Warning 5"	M 110.4	BOOL
"Warning 6"	M 110.5	BOOL
"Warning 7"	M 110.6	BOOL
"Warning 8"	M 110.7	BOOL
"Warning Activo"	M 111.0	BOOL
"Warning 9"	M 111.1	BOOL
"Hab_Rueda_Almac"	M 112.0	BOOL
"Hab_Rueda_2?"	M 112.1	BOOL
"Hab_Almacenes"	M 112.2	BOOL
"Araña_Inicializada"	M 112.3	BOOL	// Araña en Condiciones Iniciales
"INIC_Araña"	M 112.4	BOOL
"Forz_ArañaRolos"	M 113.0	BOOL
"Forz_RolosPerf"	M 113.1	BOOL
"Forz_PerfCinta"	M 113.2	BOOL
"Aux_Flanco1"	M 114.0	BOOL
"AuxFlanco2"	M 114.1	BOOL
"Frz_ReinicioPinza"	M 114.3	BOOL
"AuxFP"	M 114.4	BOOL
"AuxFn"	M 115.0	BOOL
"AuxFn2"	M 115.1	BOOL
"S_PL_0"	M 150.0	BOOL	// Plegadora - Estado 0: REINICIO
"S_PL_1"	M 150.1	BOOL	// Plegadora - Estado 1: POSICIONAR EN RECEPCIÓN
"S_PL_2"	M 150.2	BOOL	// Plegadora - Estado 2: INGRESO DE PIEZA
"S_PL_3"	M 150.3	BOOL	// Plegadora - Estado 3: POSICIONAR PLEGADO 1
"S_PL_4"	M 150.4	BOOL	// Plegadora - Estado 4: PLEGADO 1
"S_PL_5"	M 150.5	BOOL	// Plegadora - Estado 5: PLEGADO 2
"S_PL_6"	M 150.6	BOOL	// Plegadora - Estado 6: ENTREGA PIEZA
"S_PL_7"	M 150.7	BOOL	// Plegadora - Estado 7:
"S_PL_8"	M 151.0	BOOL	// Plegadora - Estado 8:
"S_PL_9"	M 151.1	BOOL	// Plegadora - Estado 9: ALINEACIÓN
"S_PL_10"	M 151.2	BOOL	// Plegadora - Estado 10: POSICIONAR PLEGADO  2
"S_PL_11"	M 151.3	BOOL	// Plegadora - Estado 11: POSICIONAR ENTREGA
"S_PL_12"	M 151.4	BOOL	// Plegadora - Estado 12: POSICIONAR ESPERA
"S_PL_13"	M 151.5	BOOL	// Plegadora - Estado 13:
"S_PL_14"	M 151.6	BOOL	// Plegadora - Estado 14:
"S_PL_15"	M 151.7	BOOL	// Plegadora - Estado 15:
"C_PL_0"	M 152.0	BOOL	// Plegadora - Contatenadora 0
"C_PL_1"	M 152.1	BOOL	// Plegadora - Contatenadora 1
"C_PL_2"	M 152.2	BOOL	// Plegadora - Contatenadora 2
"C_PL_3"	M 152.3	BOOL	// Plegadora - Contatenadora 3
"C_PL_4"	M 152.4	BOOL	// Plegadora - Contatenadora 4
"C_PL_5"	M 152.5	BOOL	// Plegadora - Contatenadora 5
"C_PL_6"	M 152.6	BOOL	// Plegadora - Contatenadora 6
"C_PL_7"	M 152.7	BOOL	// Plegadora - Contatenadora 7
"C_PL_8"	M 153.0	BOOL	// Plegadora - Contatenadora 8
"C_PL_9"	M 153.1	BOOL	// Plegadora - Contatenadora 9
"C_PL_10"	M 153.2	BOOL	// Plegadora - Contatenadora 10
"C_PL_11"	M 153.3	BOOL	// Plegadora - Contatenadora 11
"C_PL_12"	M 153.4	BOOL	// Plegadora - Contatenadora 12
"C_PL_13"	M 153.5	BOOL	// Plegadora - Contatenadora 13
"C_PL_14"	M 153.6	BOOL	// Plegadora - Contatenadora 14
"C_PL_15"	M 153.7	BOOL	// Plegadora - Contatenadora 15
"P_PL_0"	M 154.0	BOOL	// Plegadora - Prioritaria 0
"P_PL_1"	M 154.1	BOOL	// Plegadora - Prioritaria 1
"P_PL_2"	M 154.2	BOOL	// Plegadora - Prioritaria 2
"P_PL_3"	M 154.3	BOOL	// Plegadora - Prioritaria 3
"P_PL_4"	M 154.4	BOOL	// Plegadora - Prioritaria 4
"P_PL_5"	M 154.5	BOOL	// Plegadora - Prioritaria 5
"P_PL_6"	M 154.6	BOOL	// Plegadora - Prioritaria 6
"P_PL_7"	M 154.7	BOOL	// Plegadora - Prioritaria 7
"P_PL_8"	M 155.0	BOOL	// Plegadora - Prioritaria 8
"P_PL_9"	M 155.1	BOOL	// Plegadora - Prioritaria 9
"P_PL_10"	M 155.2	BOOL	// Plegadora - Prioritaria 10
"P_PL_11"	M 155.3	BOOL	// Plegadora - Prioritaria 11
"P_PL_12"	M 155.4	BOOL	// Plegadora - Prioritaria 12
"P_PL_13"	M 155.5	BOOL	// Plegadora - Prioritaria 13
"P_PL_14"	M 155.6	BOOL	// Plegadora - Prioritaria 14
"P_PL_15"	M 155.7	BOOL	// Plegadora - Prioritaria 15
"PL_Alineado_Si"	M 165.0	BOOL
"PL_Alineado_No"	M 165.1	BOOL
"PL_Cepillos_Si"	M 165.2	BOOL
"PL_Cepillos_No"	M 165.3	BOOL
"PL_Prensas_Si"	M 165.4	BOOL
"PL_Prensas_No"	M 165.5	BOOL
"PL_Fijaciones_Si"	M 165.6	BOOL
"PL_FIjaciones_No"	M 165.7	BOOL
"PL_Plegado1_Si"	M 166.0	BOOL
"PL_Plegado1_No"	M 166.1	BOOL
"PL_Plegado2_Si"	M 166.2	BOOL
"PL_Plegado2_No"	M 166.3	BOOL
"PL_Tenaza_Adentro"	M 166.4	BOOL
"PL_Avanzar_Tenaza_B"	M 167.3	BOOL	// BUSQUEDA -  Avanzar Tenaza
"PL_Retroceder_Tenaza_R"	M 167.4	BOOL	// RECEPCIÓN - Retroceder Tenaza
"PL_Cerrar_Tenaza_R"	M 167.5	BOOL	// RECEPCIÓN - Cerrar Tenaza
"PL_Abrir_Tenaza_B"	M 167.6	BOOL	// BUSQUEDA - Abrir Tenaza
"PL_Subir_Tenaza_B"	M 167.7	BOOL	// BUSQUEDA - Subir Tenaza
"PL_Bajar_Tenaza_R"	M 168.0	BOOL	// RECEPCIÓN - Bajar Tenaza
"PL_Avanzar_Tenaza_E"	M 168.1	BOOL	// ENTREGA - Avanzar Tenaza
"PL_Retroceder_Tenaza_E"	M 168.2	BOOL	// ENTREGA - Retroceder Tenaza
"PL_Cerrar_Tenaza_E"	M 168.3	BOOL	// ENTREGA - Bajar Tenaza
"PL_Abrir_Tenaza_E"	M 168.4	BOOL	// ENTREGA - Abrir Tenaza
"PL_Subir_Tenaza_E"	M 168.5	BOOL	// ENTREGA - Subir Tenaza
"PL_Bajar_Tenaza_E"	M 168.6	BOOL	// ENTREGA - Bajar Tenaza
"PL_Tenaza_Afuera"	M 168.7	BOOL
"PL_Subir_Cepillos"	M 169.0	BOOL	// BUSQUEDA - Subir Cepillos
"PL_Bajar_Cepillos"	M 169.1	BOOL	// RECEPCIÓN - Bajar Cepillos
"PL_Abrir_Tenaza_R2"	M 169.2	BOOL	// RECEPCIÓN - Abrir Tenaza 2
"PL_Alinear"	M 169.3	BOOL	// ALINEACIÓN - Alinear
"PL_Bloquear"	M 169.4	BOOL	// Bloquear para Plegado 1 (EST 4)
"PL_Bloquear2"	M 169.5	BOOL	// Bloquear para Plegado 2 (EST 5)
"PL_Desbloquear"	M 169.6	BOOL
"PL_Desbloquear2"	M 169.7	BOOL
"PL_Cerrar_Tenaza2"	M 170.0	BOOL	// ALINEACIÓN - Cerrar Tenaza
"PL_Plegar1"	M 170.1	BOOL
"PL_Plegar2"	M 170.2	BOOL
"PL_Plegadores_Bajos"	M 170.3	BOOL
"PL_Posición_Busqueda"	M 170.4	BOOL
"PL_Tenaza_Arriba"	M 170.5	BOOL
"PL_Tenaza_Abajo"	M 170.6	BOOL
"PL_Tenaza_Abierta"	M 170.7	BOOL
"PL_Tenaza_Cerrada"	M 171.0	BOOL
"PL_Tenaza_Adelante"	M 171.1	BOOL
"PL_Tenaza_Atras"	M 171.2	BOOL
"PL_Descargador_Adelante"	M 171.3	BOOL
"PL_Descargador_Atrás"	M 171.4	BOOL
"PL_Abrir_Tenaza_E2"	M 171.5	BOOL
"PL_Posición_Espera"	M 180.0	BOOL	// Ultimo Posicionamiento: Espera
"PL_Posición_Recepción"	M 180.1	BOOL	// Ultimo Posicionamiento: Recepción
"PL_Posición_Alineación"	M 180.2	BOOL	// Ultimo Posicionamiento: Alineación
"PL_Posición_Plegado1"	M 180.3	BOOL	// Ultimo Posicionamiento: Plegado 1
"PL_Posición_Plegado2"	M 180.4	BOOL	// Ultimo Posicionamiento: Plegado 2
"PL_Posición_Entrega"	M 180.5	BOOL	// Ultimo Posicionamiento: Entrega
"PL_Tenaza_AvanceSeguro"	M 180.6	BOOL
"Carga_Receta_Almacén1"	M 180.7	BOOL	// Orden de carga de receta en almacén 1
"Carga_Receta_Almacén2"	M 181.0	BOOL	// Orden de carga de receta en almacén 2
"PL_Mov_Seguro_Servos"	M 181.1	BOOL
"PI_Mov_Seguro_Servo"	M 181.2	BOOL
"PL_PPleg"	M 181.3	BOOL	// Permiso Plegado
"Aux_CerrarTenaza"	M 190.0	BOOL	// Anticipación cierre Tenaza
"PL_Anticip_Prensas"	M 190.1	BOOL	// Anticipar Bajada de prensas (EST 9)
"PL_AnticSubidaFij"	M 190.2	BOOL	// Anticipar subida Fijaciones (EST 9/3/10)
"HAB_ANTIC_FIJACIONES"	M 190.3	BOOL
"HAB_ANTIC_PRENSAS"	M 190.4	BOOL
"S_F_0"	M 204.0	BOOL	// Formador - Estado 0: DETENIDO
"S_F_1"	M 204.1	BOOL	// Formador - Estado 1: ESPERA
"S_F_2"	M 204.2	BOOL	// Formador - Estado 2: FORMADO Esquina 1 Herramienta 1
"S_F_3"	M 204.3	BOOL	// Formador - Estado 3: FORMADO Esquina 1 Herramienta 2
"S_F_4"	M 204.4	BOOL	// Formador - Estado 4: FORMADO Esquina 2 Herramienta 1
"S_F_5"	M 204.5	BOOL	// Formador - Estado 5: FORMADO Esquina 2 Herramienta 2
"S_F_6"	M 204.6	BOOL	// Formador - Estado 6: ENTREGA
"S_F_7"	M 204.7	BOOL	// Formador - Estado 7: Posiciona en Esquina 1 Herramienta 1
"S_F_8"	M 205.0	BOOL	// Formador - Estado 8: Posiciona en Esquina 1 Herramienta 2
"S_F_9"	M 205.1	BOOL	// Formador - Estado 9: Posiciona enEsquina 2 Herramienta 1
"S_F_10"	M 205.2	BOOL	// Formador - Estado 10: Posiciona en Esquina 2 Herramienta 2
"S_F_11"	M 205.3	BOOL	// Formador - Estado 11: Posiciona en Entrega
"S_F_12"	M 205.4	BOOL	// Formador - Estado 12: Posiciona en Recepción
"S_F_13"	M 205.5	BOOL	// Formador - Estado 13:
"S_F_14"	M 205.6	BOOL	// Formador - Estado 14:
"S_F_15"	M 205.7	BOOL	// Formador - Estado 15:
"C_F_0"	M 206.0	BOOL	// Formador - Contatenadora 0
"C_F_1"	M 206.1	BOOL	// Formador - Contatenadora 1
"C_F_2"	M 206.2	BOOL	// Formador - Contatenadora 2
"C_F_3"	M 206.3	BOOL	// Formador - Contatenadora 3
"C_F_4"	M 206.4	BOOL	// Formador - Contatenadora 4
"C_F_5"	M 206.5	BOOL	// Formador - Contatenadora 5
"C_F_6"	M 206.6	BOOL	// Formador - Contatenadora 6
"C_F_7"	M 206.7	BOOL	// Formador - Contatenadora 7
"C_F_8"	M 207.0	BOOL	// Formador - Contatenadora 8
"C_F_9"	M 207.1	BOOL	// Formador - Contatenadora 9
"C_F_10"	M 207.2	BOOL	// Formador - Contatenadora 10
"C_F_11"	M 207.3	BOOL	// Formador - Contatenadora 11
"C_F_12"	M 207.4	BOOL	// Formador - Contatenadora 12
"C_F_13"	M 207.5	BOOL	// Formador - Contatenadora 13
"C_F_14"	M 207.6	BOOL	// Formador - Contatenadora 14
"C_F_15"	M 207.7	BOOL	// Formador - Contatenadora 15
"P_F_0"	M 208.0	BOOL	// Formador - Prioritaria 0
"P_F_1"	M 208.1	BOOL	// Formador - Prioritaria 1
"P_F_2"	M 208.2	BOOL	// Formador - Prioritaria 2
"P_F_3"	M 208.3	BOOL	// Formador - Prioritaria 3
"P_F_4"	M 208.4	BOOL	// Formador - Prioritaria 4
"P_F_5"	M 208.5	BOOL	// Formador - Prioritaria 5
"P_F_6"	M 208.6	BOOL	// Formador - Prioritaria 6
"P_F_7"	M 208.7	BOOL	// Formador - Prioritaria 7
"P_F_8"	M 209.0	BOOL	// Formador - Prioritaria 8
"P_F_9"	M 209.1	BOOL	// Formador - Prioritaria 9
"P_F_10"	M 209.2	BOOL	// Formador - Prioritaria 10
"P_F_11"	M 209.3	BOOL	// Formador - Prioritaria 11
"P_F_12"	M 209.4	BOOL	// Formador - Prioritaria 12
"P_F_13"	M 209.5	BOOL	// Formador - Prioritaria 13
"P_F_14"	M 209.6	BOOL	// Formador - Prioritaria 14
"P_F_15"	M 209.7	BOOL	// Formador - Prioritaria 15
"Err_C_F"	M 210.0	BOOL	// Error Concatenadoras Máquina de Estados Formador
"Err_P_F"	M 210.1	BOOL	// Error Prioritarias Máquina de Estados Formador
"F_ActivarH1_E1"	M 210.2	BOOL	// Activar Herramienta 1 (Esquina 1)
"F_ActivarH1_E2"	M 210.3	BOOL	// Activar Herramienta 1 (Esquina 2)
"F_ActivarH2_E1"	M 210.4	BOOL	// Activar Herramienta 2 (Esquina 1)
"F_ActivarH2_E2"	M 210.5	BOOL	// Activar Herramienta 2 (Esquina 2)
"F_H1_Activada"	M 210.6	BOOL
"F_H1_Desactivada"	M 210.7	BOOL
"F_H2_Activada"	M 211.0	BOOL
"F_H2_Desactivada"	M 211.1	BOOL
"F_H_Arriba"	M 211.2	BOOL
"F_H_Abajo"	M 211.3	BOOL
"F_H1_Matriz_SI"	M 211.4	BOOL
"F_H1_Matriz_NO"	M 211.5	BOOL
"F_H1_Martillo_SI"	M 211.6	BOOL
"F_H1_Martillo_NO"	M 211.7	BOOL
"F_H2_Matriz_SI"	M 212.0	BOOL
"F_H2_Matriz_NO"	M 212.1	BOOL
"F_H2_Martillo_SI"	M 212.2	BOOL
"F_H2_Martillo_NO"	M 212.3	BOOL
"F_H1_Ciclo_FIN"	M 212.4	BOOL
"F_H2_Ciclo_FIN"	M 212.5	BOOL
"F_TTH1"	M 212.6	BOOL	// Trabajo Terminado Herramienta 1
"F_TTH2"	M 212.7	BOOL	// Trabajo Terminado Herramienta 2
"PL_INIC"	M 213.0	BOOL	// Inicialización Automática de Plegadores
"PI_INIC"	M 213.1	BOOL	// Inicialización Automática de Pinza
"PL_INIC_AP_OK"	M 213.2	BOOL	// Inicialización Automática de Plegadores Apertura Lista
"PL_INIC_AP"	M 213.3	BOOL	// Inicialización Automática de Plegadores Apertura
"PI_INIC_OP"	M 213.4	BOOL	// Solicitud de Inicialización de Pinza Operador
"PL_Mov_Hid"	M 220.0	BOOL	// Movimiento hidráulico en plegadora
"PL_Mov_Neum"	M 220.1	BOOL	// Movimiento Neumático en Plegadora
"PL_Mov_Desc"	M 220.2	BOOL	// Movimiento de Descargador
"CLIGNO"	MB 9	BYTE
"IM14"	MB 40	BYTE	// image carte 14
"T_Parcial_H"	MD 120	REAL	// Tiempo Parcial Heladera
"T_H_P"	MD 124	REAL	// Tiempo Heladera Previo
"Hel_x_H"	MD 128	REAL	// Heladeras por Hora
"Hel_x_Min"	MD 132	REAL	// Heladeras por Minuto
"T_Helad"	MD 136	REAL	// Tiempo Instantáneo Heladera
"Prom_T_HEL"	MD 140	REAL	// Tiempo Promedio por Heladera
"T_Hel_Tend"	MD 144	REAL	// Tendencia de Tiempo x Heladera
"Cant_Prom"	MD 160	REAL	// Cantidad de Heladeras para Promedio
"ProD"	MD 200	DINT
"Error_Pinza_Ant_Rec"	MD 230	DWORD
"Error_Pinza_Ant_E1H1"	MD 234	DWORD
"Error_Pinza_Ant_E1H2"	MD 238	DWORD
"Error_Pinza_Ant_E2H1"	MD 242	DWORD
"Error_Pinza_Ant_E2H2"	MD 246	DWORD
"Error_Pinza_Ant_Ent"	MD 250	DWORD
"RC1_VAL"	MW 30	INT	// Rueda 1
"RC2_VAL"	MW 32	INT	// Rueda 2
"W_S_PL"	MW 150	WORD	// Estados Plegadora
"W_C_PL"	MW 152	WORD	// Concatenadoras Plegadora
"W_P_PL"	MW 154	WORD	// Prioritarias Plegadora
"RET_VAL"	MW 160	INT
"W_S_F"	MW 204	WORD	// Estados Formador
"W_C_F"	MW 206	WORD	// Concatenadoras Formador
"W_P_F"	MW 208	WORD	// Prioritarias Formador
"I/O_FLT1"	OB 82	OB 82	// I/O Point Fault 1
"RACK_FLT"	OB 86	OB 86	// Loss of Rack Fault
"COMPLETE RESTART"	OB 100	OB 100	// Complete Restart
"PROG_ERR"	OB 121	OB 121	// Programming Error
"MOD_ERR"	OB 122	OB 122	// Module Access Error
"KM05"	Q 0.0	BOOL	// Perfilador Marcha Bombas de Lubricación
"KM06"	Q 0.1	BOOL	// Perfilador Marcha Grupo Hidráulico Freno
"KM07.1"	Q 0.2	BOOL	// Avance Ajuste de Ancho Perfilador
"KM07.2"	Q 0.3	BOOL	// Retroceso Ajuste de Ancho Perfilador
"KM09.1"	Q 0.4	BOOL	// Avance Ajuste de Formado
"KM09.2"	Q 0.5	BOOL	// Retroceso Ajuste de Formado
"KM13.1"	Q 0.6	BOOL	// Plegadora Marcha Grupo Hidráulico
"KM14"	Q 0.7	BOOL	// Encendido Calentador de Chapa
"KM13.2"	Q 1.0	BOOL	// Plegadora Marcha Refrigerador Grupo Hidráulico
"40Y1"	Q 1.1	BOOL	// Válvula Aire a Tulipas - Grupo 1
"40Y2"	Q 1.2	BOOL	// Válvula Aire a Tulipas - Grupo 2
"40Y3"	Q 1.3	BOOL	// Válvula Aire a Tulipas - Grupo 3
"40Y4"	Q 1.4	BOOL	// Válvula Vacío a Tulipas - Grupo 1
"40Y5"	Q 1.5	BOOL	// Válvula Vacío a Tulipas - Grupo 2
"40Y6"	Q 1.6	BOOL	// Válvula Vacío a Tulipas - Grupo 3
"40Y7"	Q 1.7	BOOL	// Araña - Subir (Pistón Inferior)
"41Y1"	Q 2.0	BOOL	// Araña -  Bajar (Pistón Inferior)
"41Y2"	Q 2.1	BOOL	// Araña - Bajar (Pistón Superior)
"41Y3"	Q 2.2	BOOL	// Araña -  Subir (Pistón Superior)
"VAR02_RUN"	Q 2.3	BOOL	// Transporte Araña en Funcionamiento
"KM02_1"	Q 2.4	BOOL	// Avance Transporte de Araña
"KM02_2"	Q 2.5	BOOL	// Retroceso Transporte de Araña
"VAR03_RUN"	Q 2.6	BOOL	// Marcha Transporte Rolos
"VAR03_RC"	Q 2.7	BOOL	// Marcha Invertida Transporte Rolos
"42K1"	Q 3.0	BOOL	// Desbloqueo Freno Perfilador
"42K2"	Q 3.1	BOOL	// Plegadora ByPass Grupo áulico
"42K3"	Q 3.2	BOOL	// Formador Herramienta 1 - Accionar Martillo
"42K4"	Q 3.3	BOOL	// Formador Herramienta 1 - Liberar Martillo
"42K5"	Q 3.4	BOOL	// Formador Herramienta 1 - Accionar Martiz
"42K6"	Q 3.5	BOOL	// Formador Herramienta 1 - Liberar Martiz
"42K7"	Q 3.6	BOOL	// Formador Herramienta 2 - Accionar Martillo
"42K8"	Q 3.7	BOOL	// Formador Herramienta 2 - Liberar Martillo
"43K1"	Q 4.0	BOOL	// Formador Herramienta 2 - Accionar Martiz
"43K2"	Q 4.1	BOOL	// Formador Herramienta 2 - Liberar Martiz
"43K3"	Q 4.2	BOOL	// Formador Bloquear Herramienta
"43K4"	Q 4.3	BOOL	// Formador Desbloquear Herramienta
"43Y5"	Q 4.4	BOOL	// Liberar Parada Formador
"43Y6"	Q 4.5	BOOL	// Accionar Parada Formador
"43Y7"	Q 4.6	BOOL	// Abir Pinza
"43Y8"	Q 4.7	BOOL	// Cerrar Pinza
"44Y1"	Q 5.0	BOOL	// Tenaza Plegadora Avance
"44Y2"	Q 5.1	BOOL	// Tenaza Plegadora Retroceso
"44Y3"	Q 5.2	BOOL	// Tenaza Plegadora Bajar
"44Y4"	Q 5.3	BOOL	// Tenaza Plegadora Subir
"44Y5"	Q 5.4	BOOL	// Tenaza Plegadora Abrir
"44Y6"	Q 5.5	BOOL	// Tenaza Plegadora Cerrar
"VAR08_RUN"	Q 5.6	BOOL	// Avance Transporte Cinta
"VAR08_RC"	Q 5.7	BOOL	// Retroceso Transporte Cinta
"45K1"	Q 6.0	BOOL	// Avanzar Descargador
"45K2"	Q 6.1	BOOL	// Retroceder Descargador
"45K3"	Q 6.2	BOOL	// Plegador 1 Avance Fijación
"45K4"	Q 6.3	BOOL	// Plegador 1 Retroceso Fijación
"45K5"	Q 6.4	BOOL	// Plegador 1 Subir
"45K6"	Q 6.5	BOOL	// Plegador 1 Bajar
"45K7"	Q 6.6	BOOL	// Subir Prensa Plegador 1
"45K8"	Q 6.7	BOOL	// Bajar Prensa Plegador 1
"46K1"	Q 7.0	BOOL	// Subir Extención 1 Prensa Plegador 1
"46K2"	Q 7.1	BOOL	// Bajar Extención 1 Prensa Plegador 1
"46K3"	Q 7.2	BOOL	// Subir Extención 2 Prensa Plegador 1
"46K4"	Q 7.3	BOOL	// Bajar Extención 2 Prensa Plegador 1
"46K5"	Q 7.4	BOOL	// Plegadora Alineadores X
"46K6"	Q 7.5	BOOL	// Plegadora Alineadores Y
"46K7"	Q 7.6	BOOL	// Plegadora Subir Cepillos
"46K8"	Q 7.7	BOOL	// Desbloqueo Freno Ajuste de Formado
"47K1"	Q 8.0	BOOL	// Plegador 2 Avance Fijación
"47K2"	Q 8.1	BOOL	// Plegador 2 Retroceso Fijación
"47K3"	Q 8.2	BOOL	// Plegador 2 Subir
"47K4"	Q 8.3	BOOL	// Plegador 2 Bajar
"47K5"	Q 8.4	BOOL	// Subir Prensa Plegador 2
"47K6"	Q 8.5	BOOL	// Bajar Prensa Plegador 2
"47K7"	Q 8.6	BOOL	// Subir Extención 1 Prensa Plegador 2
"47K8"	Q 8.7	BOOL	// Bajar Extención 1 Prensa Plegador 2
"48K1"	Q 9.0	BOOL	// Subir Extención 2 Prensa Plegador 2
"48K2"	Q 9.1	BOOL	// Bajar Extención 2 Prensa Plegador 2
"oHomming"	Q 9.2	BOOL	// Lámpara Homming realizado
"PH_Sel_P1"	Q 9.3	BOOL	// Habilitar Fin de Carrera Araña 1
"PH_Sel_P2"	Q 9.4	BOOL	// Habilitar Fin de Carrera Araña 2
"PH_Sel_P3"	Q 9.5	BOOL	// Habilitar Fin de Carrera Araña 3
"Reserva10"	Q 9.6	BOOL	// Reserva
"oVlvHabPresForm"	Q 9.7	BOOL	// Válvula Hab Presión Formador
"PRF_SLM_DATA14"	Q 24.0	BOOL
"PRF_SLM_PLC"	Q 24.1	BOOL	// SmartLine Perfiladora Mando PLC
"PRF_SLM_DATA15"	Q 24.2	BOOL
"PRF_SLM_DATA16"	Q 24.3	BOOL
"PRF_SLM_DATA17"	Q 24.4	BOOL
"PRF_SLM_DATA18"	Q 24.5	BOOL
"PRF_SLM_DATA19"	Q 24.6	BOOL
"PRF_SLM_DATA20"	Q 24.7	BOOL
"PRF_SLM_CON_DES1"	Q 25.0	BOOL	// SmartLine Perfiladora CON/DES 1 Infeed
"PRF_SLM_DES2"	Q 25.1	BOOL	// SmartLine Perfiladora DES 2 Infeed
"PRF_SLM_DATA11"	Q 25.2	BOOL
"PRF_SLM_HS"	Q 25.3	BOOL	// SmartLine Perfiladora Habilitar Servicio
"PRF_SLM_DATA12"	Q 25.4	BOOL
"PRF_SLM_DATA13"	Q 25.5	BOOL
"PRF_SLM_BA"	Q 25.6	BOOL	// SmartLine Perfiladora Bloquear Alimentación
"PRF_SLM_CF"	Q 25.7	BOOL	// SmartLine Perfiladora Confirmar Fallos
"PRF_DATA12"	Q 26.0	BOOL
"PRF_DATA13"	Q 26.1	BOOL
"PRF_SC"	Q 26.2	BOOL	// Perfiladora Suprimir Confirmación Automáticamente
"PRF_DATA14"	Q 26.3	BOOL
"PRF_DATA15"	Q 26.4	BOOL
"PRF_DATA16"	Q 26.5	BOOL
"PRF_DATA17"	Q 26.6	BOOL
"PRF_DATA18"	Q 26.7	BOOL
"PRF_SS"	Q 27.0	BOOL	// Perfiladora Detector Señal de Sincronización
"PRF_RTC"	Q 27.1	BOOL	// Perfiladora RTC Sincronización en Tiempo Real
"PRF_PERF1_DES3"	Q 27.2	BOOL	// Perfiladora Drive 1 DES3
"PRF_PERF2_DES3"	Q 27.3	BOOL	// Perfiladora Drive 2 DES3
"PRF_PERF3_DES3"	Q 27.4	BOOL	// Perfiladora Drive 3 DES3
"PRF_PERF4_DES3"	Q 27.5	BOOL	// Perfiladora Drive 4 DES3
"PRF_CTF"	Q 27.6	BOOL	// Perfiladora Confirmar Todos los Fallos
"PRF_CF"	Q 27.7	BOOL	// Perfiladora Confirmar Fallos
"COD1_INIT"	Q 40.7	BOOL	// Perfilador Consigna Inicio
"COD2_INIT"	Q 44.7	BOOL	// Formador Consigna Inicio
"VAR_02_Acquit"	Q 51.7	BOOL	// Reconocer Fallos Variador Araña
"VAR_03_Acquit"	Q 54.7	BOOL	// Reconocer Fallos Variador Transporte Rolos
"VAR_08_Acquit"	Q 59.7	BOOL	// Reconocer Fallos Variador Cinta Transpore
"PL1_jg-"	Q 62.0	BOOL	// Plegador 1 Jog Retroceso
"PL1_jg+"	Q 62.1	BOOL	// Plegador 1 Jog Avance
"PL1_vie"	Q 62.2	BOOL	// Plegador 1 Bit de Vida
"PL1_reference"	Q 62.3	BOOL	// Plegador 1 Referenciar
"Ref_PL1"	Q 62.4	BOOL	// Solicitud de referenciado del PL1
"PL1_DDS"	Q 62.5	BOOL	// Plegador 1 DDS (0=encoder, 1=regla)
"PL1_on"	Q 63.0	BOOL	// Plegador 1 Con/Des
"PL1_arret2"	Q 63.1	BOOL	// Plegador 1 Des2
"PL1_arret3"	Q 63.2	BOOL	// Plegador 1 Des3
"PL1_lib"	Q 63.3	BOOL	// Plegador 1 Habilitar Sevicio
"PL1_rj"	Q 63.4	BOOL	// Plegador 1 Desechar petición de Desplazamiento
"PL1_stop"	Q 63.5	BOOL	// Plegador 1 Parada
"PL1_start"	Q 63.6	BOOL	// Plegador 1 Activar Petición de Desplazamiento
"PL1_reset"	Q 63.7	BOOL	// Plegador 1 Confirmar Fallos
"PL1_Jog"	Q 67.1	BOOL
"PL1_Hab_Regla_Balluff"	Q 69.0	BOOL	// PL1: Habilita la regla Balluff como sist. de medida usado para el ctrl de pos.
"PL2_jg-"	Q 82.0	BOOL	// Plegador 2 Jog Retroceso
"PL2_jg+"	Q 82.1	BOOL	// Plegador 2 Jog Avance
"PL2_vie"	Q 82.2	BOOL	// Plegador 2 Bit de Vida
"PL2_reference"	Q 82.3	BOOL	// Plegador 2 Referenciar
"Ref_PL2"	Q 82.4	BOOL	// Solicitud de referenciado del PL2
"PL2_DDS"	Q 82.5	BOOL	// Plegador 2 DDS (0=encoder, 1=regla)
"PL2_on"	Q 83.0	BOOL	// Plegador 2 Con/Des
"PL2_arret2"	Q 83.1	BOOL	// Plegador 2 Des2
"PL2_arret3"	Q 83.2	BOOL	// Plegador 2 Des3
"PL2_lib"	Q 83.3	BOOL	// Plegador 2 Habilitar Sevicio
"PL2_rj"	Q 83.4	BOOL	// Plegador 2 Desechar petición de Desplazamiento
"PL2_stop"	Q 83.5	BOOL	// Plegador 2 Parada
"PL2_start"	Q 83.6	BOOL	// Plegador 2 Activar Petición de Desplazamiento
"PL2_reset"	Q 83.7	BOOL	// Plecador 2 Confirmar Fallos
"PL2_Jog"	Q 87.1	BOOL
"PL2_Hab_Regla_Balluff"	Q 89.0	BOOL	// PL2: Habilita la regla Balluff como sist. de medida usado para el ctrl de pos.
"PI_jg-"	Q 102.0	BOOL	// Pinza Jog Retroceso
"PI_jg+"	Q 102.1	BOOL	// Pinza Jog Avance
"PI_vie"	Q 102.2	BOOL	// Pinza Bit de vida
"PI_reference"	Q 102.3	BOOL	// Pinza Referenciar
"CU_PL_Reset"	Q 102.4	BOOL	// CU Plegadora - Confirmar fallos
"PI_on"	Q 103.0	BOOL	// Pinza Con/Des
"PI_arret2"	Q 103.1	BOOL	// Pinza Des2
"PI_arret3"	Q 103.2	BOOL	// Pinza Des3
"PI_lib"	Q 103.3	BOOL	// Pinza Habilitar Servicio
"PI_rj"	Q 103.4	BOOL	// Pinza Desechar petición de Desplazamiento
"PI_stop"	Q 103.5	BOOL	// Pinza Parada
"PI_start"	Q 103.6	BOOL	// Pinza Activar Petición de Desplazamiento
"PI_reset"	Q 103.7	BOOL	// Pinza Confirmar Fallos
"PLinza_Hab_Regla_Balluff"	Q 109.0	BOOL	// Pinza: Habilita la regla Balluff como sist. de medida usado para el ctrl de pos
"18SH1"	Q 124.0	BOOL	// Lámpara En servicio
"37H1"	Q 124.1	BOOL	// Lámpara Automático
"21H1"	Q 124.2	BOOL	// Lámpara En Ciclo
"37H2"	Q 124.3	BOOL	// Lámpara Verde
"37H3"	Q 124.4	BOOL	// Lámpara Azul
"37H4"	Q 124.5	BOOL	// Lámpara Roja
"37CT1"	Q 124.6	BOOL	// Contador Horas de Marcha
"RecFallas"	Q 124.7	BOOL	// Reconocer Fallas
"KM01_1"	Q 125.0	BOOL	// Avance Intercambiador de Almacenes
"KM01_2"	Q 125.1	BOOL	// Retroceso Intercambiador de Almacenes
"KM04_AV"	Q 125.2	BOOL	// Avance Perfilador
"KM04_RC"	Q 125.3	BOOL	// Retroceso Perfilador
"KM04_GV"	Q 125.4	BOOL	// Velocidad Rápida Perfilador
"Reserva6"	Q 125.5	BOOL	// Reserva
"oLmp_Azul_Alm"	Q 125.6	BOOL	// Lámpara Azul Almacenes
"Reserva8"	Q 125.7	BOOL	// Reserva
"COD1_CONS"	QD 40	DINT	// Consigna Perfilador
"COD2_CONS"	QD 44	DINT	// Consigna Formador
"PL1_position"	QD 72	DINT	// Plegador 1 Consigna Posición
"PL1_vitesse"	QD 76	DINT	// Plegador 1 Consigna Velocidad
"PL2_position"	QD 92	DINT	// Plegador 2 Consigna Posición
"PL2_vitesse"	QD 96	DINT	// Plegador 2 Consigna Velocidad
"PI_position"	QD 112	DINT	// Pinza Consigna Posición
"PI_vitesse"	QD 116	DWORD	// Pinza Consigna Velocidad
"VAR_02_Commande"	QW 50	INT	// Variador Araña Control Word
"VAR_02_SP_VEL"	QW 52	INT	// Variador Araña Consigna Velocidad (16#4000 = 100%)
"VAR_03_Commande"	QW 54	INT	// Variador Transporte Rolos Control Word
"VAR_03_CVitesse"	QW 56	INT	// Variador Transporte Rolos Consigna Velocidad (16#4000 = 100%)
"VAR_08_Commande"	QW 58	INT	// Variador Cinta Transporte Control Word
"VAR_08_CVitesse"	QW 60	INT	// Variador Cinta Transporte Consigna Velocidad (16#4000 = 100%)
"PL1_mode"	QW 64	INT	// Plegador 1 Modo de Funcionamiento
"PL1_limvit"	QW 70	INT	// Plegador 1 Límite Velocidad 80% =4000
"PL2_mode"	QW 84	INT	// Plegador 2 Modo de Funcionamiento
"PL2_limvit"	QW 90	INT	// Plegador 2 Límite Velocidad 80% =4000
"PI_mode"	QW 104	INT	// Pinza Modo de Funcionamiento
"PI_limvit"	QW 110	INT	// Pinza Límite Velocidad 80% =4000
"PUT"	SFB 15	SFB 15	// Write Data to a Remote CPU
"ALARM_SQ"	SFC 17	SFC 17	// Generate Block-Related Messages with Acknowledgment
"ALARM_S"	SFC 18	SFC 18	// Generate Permanently Acknowledged Block-Related Messages
"BLKMOV"	SFC 20	SFC 20	// Copy Variables
"WR_USMSG"	SFC 52	SFC 52	// Write a User-Defined Diagnostic Event to the Diagnostic Buffer
"TIME_TCK"	SFC 64	SFC 64	// Read the System Time
"T_Reset"	T 0	TIMER	// Tiempo de reseteo de fallas
"Marcha_GH_Min"	T 1	TIMER	// Tiempo de marcha mínimo Grupo Hidráulico
"T_MES"	T 3	TIMER	// Tiempo Ajuste Tensión
"T_Agarrado"	T 5	TIMER	// Tiempo de Agarrado de Chapa (Araña)
"T_Soltado"	T 6	TIMER	// Tiempo de Soltado de Chapa (Araña)
"PI_TPOS"	T 8	TIMER	// Pinza Tiempo para Posicionamiento
"PI_TSTART"	T 9	TIMER	// Pinza Tiempo Arranque
"T_KM7_0"	T 10	TIMER
"T_Herr_Desbloq"	T 11	TIMER	// Tiempo para asegurar Herramientas Desbloqueadas
"PL1_TPOS"	T 16	TIMER	// Plegador 1 Tiempo para Posicionamiento
"PL1_TSTART"	T 17	TIMER	// Plegador 1 Tiempo Arranque
"PL2_TPOS"	T 18	TIMER	// Plegador 2 Tiempo para Posicionamiento
"PL2_TSTART"	T 19	TIMER	// Plegador 2 Tiempo Arranque
"T_AvAraña"	T 20	TIMER
"T_SubirAraña"	T 21	TIMER
"T_Avance_Pinza"	T 22	TIMER
"T_BajarTenaza"	T 23	TIMER
"T_AbrirTenaza"	T 24	TIMER
"T_ActAlinX"	T 25	TIMER
"T_ActAlinY"	T 26	TIMER
"T_SubirCepillos"	T 27	TIMER
"T_BajarAraña2"	T 29	TIMER
"T_SubirFij1"	T 30	TIMER
"T_SubirPL1"	T 31	TIMER
"T_SubirPrensaPL1"	T 32	TIMER
"T_SubirExte1PL1"	T 33	TIMER
"T_SubirExt2PL1"	T 34	TIMER
"T_SubirFij2"	T 35	TIMER
"T_SubirPL2"	T 36	TIMER
"T_SubirPrensaPL2"	T 37	TIMER
"T_SubirExt1PL2"	T 38	TIMER
"T_SubirExt2PL2"	T 39	TIMER
"T_RetAjForm"	T 40	TIMER
"T_DesbloqAvForm"	T 41	TIMER
"T_CerrarPinza"	T 42	TIMER
"T_RetDesc"	T 44	TIMER
"T_bourrage"	T 45	TIMER
"T_OnMH1"	T 50	TIMER
"T_OnMTH1"	T 51	TIMER
"T_OnMH2"	T 52	TIMER
"T_OnMTH2"	T 53	TIMER
"T_BlqH"	T 54	TIMER
"T_AvAlm"	T 55	TIMER
"T_AvDesc"	T 56	TIMER
"Alin_Y_Simu"	T 59	TIMER	// Simulación de Alineación en Y
"T_Excursión_Formador"	T 61	TIMER	// Tiempo Máximo de excursión ancho Cinta
"T_DbloqH"	T 64	TIMER
"T_RetAlm"	T 66	TIMER
"T_BajarCepillos"	T 72	TIMER
"T_Retroceso_Pinza"	T 74	TIMER
"T_SubirTenaza"	T 75	TIMER
"T_CerrarTenaza"	T 76	TIMER
"T_DesacAlinX"	T 77	TIMER
"T_DesactAlinY"	T 78	TIMER
"T_BajarFij1"	T 80	TIMER
"T_BajarPL1"	T 81	TIMER
"T_BajarPrensaPL1"	T 82	TIMER
"T_BajarExte1PL1"	T 83	TIMER
"T_BajarExt2PL1"	T 84	TIMER
"T_BajarFij2"	T 85	TIMER
"T_BajarPL2"	T 86	TIMER
"T_BajarPrensaPL2"	T 87	TIMER
"T_BajarExt1PL2"	T 88	TIMER
"T_BajarExt2PL2"	T 89	TIMER
"T_RetAraña"	T 90	TIMER
"T_BajarAraña"	T 91	TIMER
"T_SubirAraña2"	T 92	TIMER
"T_AvAjForm"	T 93	TIMER
"T_BloqueaAvForm"	T 94	TIMER
"T_AbrirPinza"	T 95	TIMER
"T_OffMH1"	T 96	TIMER
"T_OffMTH1"	T 97	TIMER
"T_OffMH2"	T 98	TIMER
"T_OffMTH2"	T 99	TIMER
"Tiempo_Warning_1"	T 100	TIMER
"Tiempo_Warning_2"	T 101	TIMER
"Tiempo_Warning_3"	T 102	TIMER
"Tiempo_Warning_4"	T 103	TIMER
"Tiempo_Warning_5"	T 104	TIMER
"Tiempo_Warning_6"	T 105	TIMER
"Tiempo_Warning_7"	T 106	TIMER
"Tiempo_Warning_8"	T 107	TIMER
"Ret_PosPL_Busqueda"	T 110	TIMER	// Retardo para envío de orden de posicionamiento de Búsqueda
"Ret_PosPL_Alineación"	T 111	TIMER	// Retardo para envío de orden de posicionamiento de Alineación
"Ret_PosPL_Plegado1"	T 112	TIMER	// Retardo para envío de orden de posicionamiento de Plegado 1
"Ret_PosPL_Plegado2"	T 113	TIMER	// Retardo para envío de orden de posicionamiento de Plegado 2
"Ret_PosPL_Entrega"	T 114	TIMER	// Retardo para envío de orden de posicionamiento de Entrega
"Ret_PosPL_Espera"	T 115	TIMER	// Retardo para envío de orden de posicionamiento de Espera
"F_T_H1"	T 116	TIMER	// Trabajo H1 Terminado
"F_T_H2"	T 117	TIMER	// Trabajo H2 Terminado
"Ret_PosF_E1H1"	T 118	TIMER	// Retardo para envío de orden de posicionamiento de Esquina 1 H1
"Ret_PosF_E1H2"	T 119	TIMER	// Retardo para envío de orden de posicionamiento de Esquina 1 H2
"Ret_PosF_E2H1"	T 120	TIMER	// Retardo para envío de orden de posicionamiento de Esquina 2 H1
"Ret_PosF_E2H2"	T 121	TIMER	// Retardo para envío de orden de posicionamiento de Esquina 2 H2
"Ret_PosF_Entrega"	T 122	TIMER	// Retardo para envío de orden de posicionamiento Entrega
"Ret_PosF_Inicial"	T 123	TIMER	// Retardo para envío de orden de posicionamiento Inicial
"T_AperturaPL1"	T 125	TIMER
"T_AperturaPL2"	T 126	TIMER
"T_Cond_Bloq1"	T 130	TIMER	// Tiempo condiciones bloqueo para PLEGADO 1
"T_Cond_Pleg1"	T 131	TIMER	// Tiempo condiciones Plegado 1
"PL_PermisoPlegado"	T 132	TIMER	// Permiso para plegado
"T_Cond_Bloq2"	T 133	TIMER	// Tiempo condiciones bloqueo para PLEGADO 2
"T_Cond_Pleg2"	T 134	TIMER	// Tiempo condiciones Plegado 2
"PL_Tiempo_Desh_AnticFij"	T 142	TIMER	// Tiempo anticipación subida fijaciones
"PL_Tiempo_AnticPren"	T 143	TIMER	// Tiempo anticipación subida prensas (EST 10/11)
"PL_Tiempo_Alineacion"	T 144	TIMER	// Tiempo para asegurar alineación
"T_Descarga"	T 164	TIMER	// Retardo Borrado de datos Descargador
"PL_Descargador_NO_Ade_T"	T 176	TIMER
"MP"	UDT 1	UDT 1	// Mot Piece
"UDT Offset"	UDT 4	UDT 4
"VAT_1"	VAT 1	
"SINAMICS"	VAT 2	
"VAT_MP"	VAT 3	
"VAT_RECETTE"	VAT 4	
"Modo_Mix"	VAT 5		// Análisis del modo mix
"VAT_DATOS_PIEZAS"	VAT 6	
"VAT_eproc"	VAT 7	
END_SYMBOL_TABLE

FUNCTION "Homing Plegadores" : VOID	// FC 1
VERSION : 0.1
BEGIN
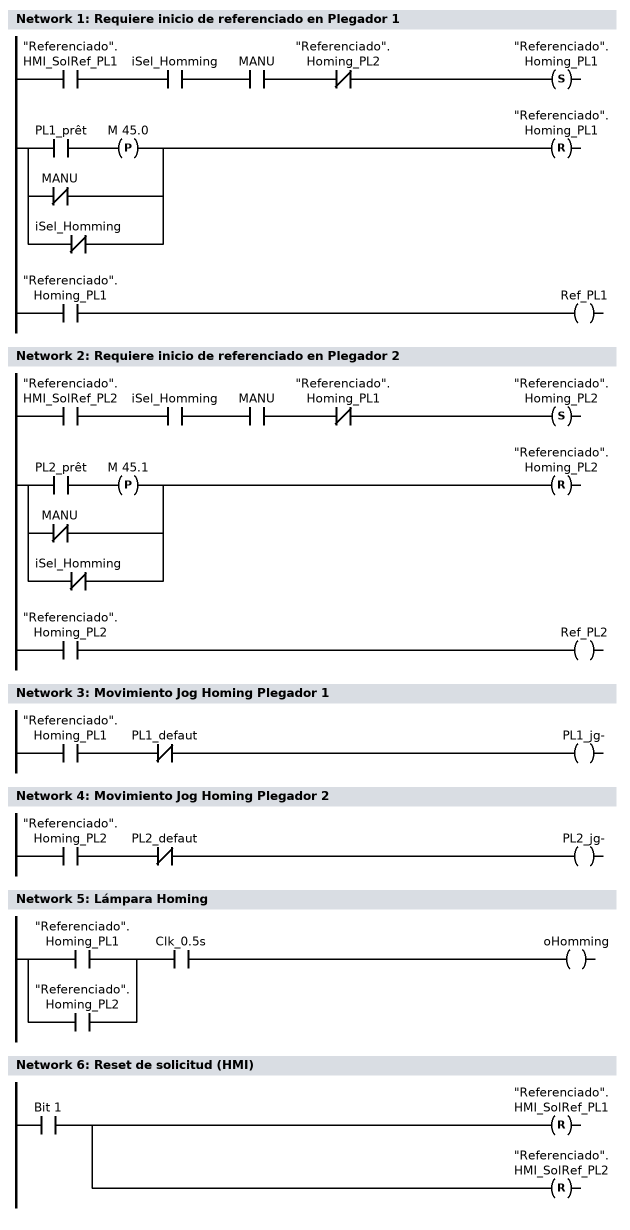
NETWORK
TITLE = Requiere inicio de referenciado en Plegador 1
      A     "Referenciado".HMI_SolRef_PL1;
      A     "iSel_Homming";
      A     "MANU";
      AN    "Referenciado".Homing_PL2;
      S     "Referenciado".Homing_PL1;
      A(;
      A     "PL1_prêt";
      FP    M 45.0;
      ON    "MANU";
      ON    "iSel_Homming";
      );
      R     "Referenciado".Homing_PL1;
      A     "Referenciado".Homing_PL1;
      =     "Ref_PL1";
NETWORK
TITLE = Requiere inicio de referenciado en Plegador 2
      A     "Referenciado".HMI_SolRef_PL2;
      A     "iSel_Homming";
      A     "MANU";
      AN    "Referenciado".Homing_PL1;
      S     "Referenciado".Homing_PL2;
      A(;
      A     "PL2_prêt";
      FP    M 45.1;
      ON    "MANU";
      ON    "iSel_Homming";
      );
      R     "Referenciado".Homing_PL2;
      A     "Referenciado".Homing_PL2;
      =     "Ref_PL2";
NETWORK
TITLE = Movimiento Jog Homing Plegador 1
      A     "Referenciado".Homing_PL1;
      AN    "PL1_defaut";
      =     "PL1_jg-";
NETWORK
TITLE = Movimiento Jog Homing Plegador 2
      A     "Referenciado".Homing_PL2;
      AN    "PL2_defaut";
      =     "PL2_jg-";
NETWORK
TITLE = Lámpara Homing
      A(;
      O     "Referenciado".Homing_PL1;
      O     "Referenciado".Homing_PL2;
      );
      A     "Clk_0.5s";
      =     "oHomming";
NETWORK
TITLE = Reset de solicitud (HMI)
      A     "Bit 1";
      R     "Referenciado".HMI_SolRef_PL1;
      R     "Referenciado".HMI_SolRef_PL2;
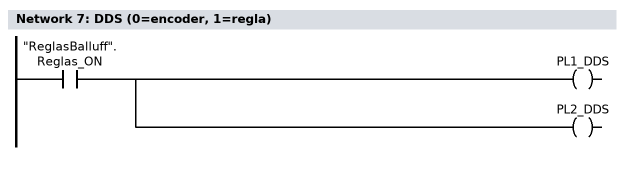
NETWORK
TITLE = DDS (0=encoder, 1=regla)
      A     "ReglasBalluff".Reglas_ON;
      =     "PL1_DDS";
      =     "PL2_DDS";
END_FUNCTION

FUNCTION "ModoMix" : VOID	// FC 2
VERSION : 0.1
BEGIN
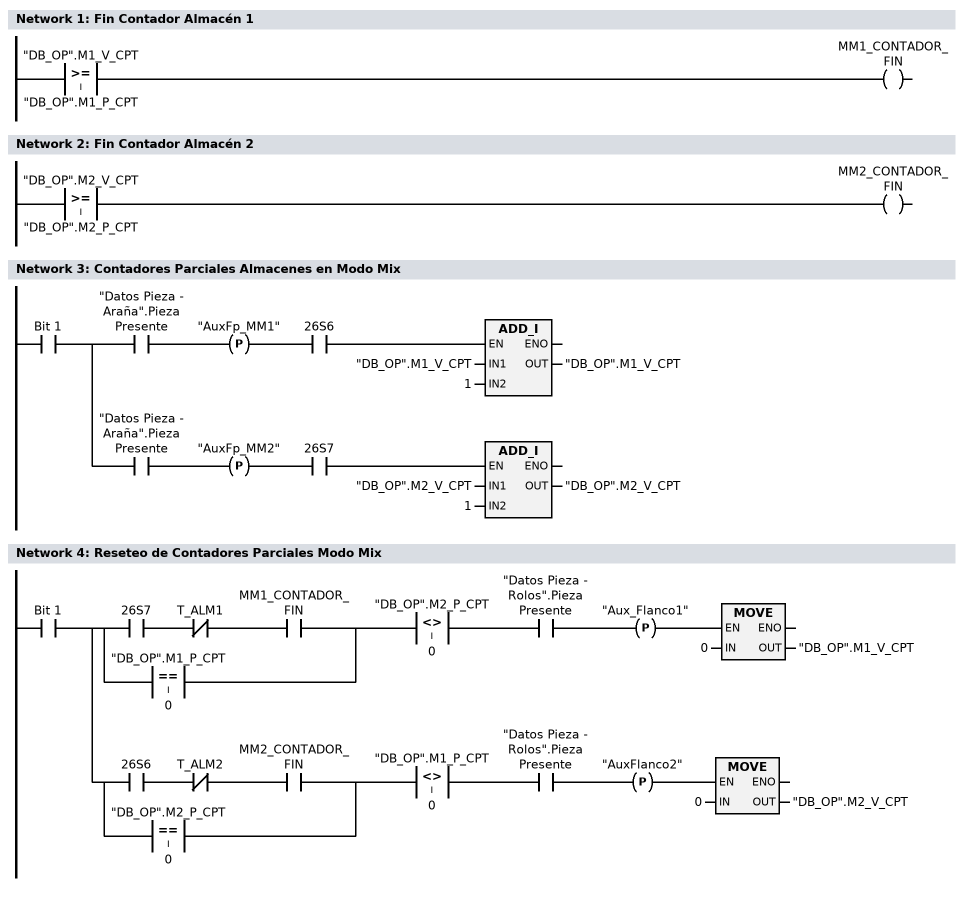
NETWORK
TITLE = Fin Contador Almacén 1
      L     "DB_OP".M1_V_CPT;
      L     "DB_OP".M1_P_CPT;
      >=I;
      =     "MM1_CONTADOR_FIN";
NETWORK
TITLE = Fin Contador Almacén 2
      L     "DB_OP".M2_V_CPT;
      L     "DB_OP".M2_P_CPT;
      >=I;
      =     "MM2_CONTADOR_FIN";
NETWORK
TITLE = Contadores Parciales Almacenes en Modo Mix
      A     "Bit 1";
      =     L 0.0;
      A     L 0.0;
      A     "Datos Pieza - Araña".PiezaPresente;
      FP    "AuxFp_MM1";
      A     "26S6";
      JNB   _001;
      L     "DB_OP".M1_V_CPT;
      L     1;
      +I;
      T     "DB_OP".M1_V_CPT;
_001: NOP   0;
      A     L 0.0;
      A     "Datos Pieza - Araña".PiezaPresente;
      FP    "AuxFp_MM2";
      A     "26S7";
      JNB   _002;
      L     "DB_OP".M2_V_CPT;
      L     1;
      +I;
      T     "DB_OP".M2_V_CPT;
_002: NOP   0;
NETWORK
TITLE = Reseteo de Contadores Parciales Modo Mix
      A     "Bit 1";
      =     L 0.0;
      A     L 0.0;
      A(;
      A     "26S7";
      AN    "T_ALM1";
      A     "MM1_CONTADOR_FIN";
      O(;
      L     "DB_OP".M1_P_CPT;
      L     0;
      ==I;
      );
      );
      A(;
      L     "DB_OP".M2_P_CPT;
      L     0;
      <>I;
      );
      A     "Datos Pieza - Rolos".PiezaPresente;
      FP    "Aux_Flanco1";
      JNB   _003;
      L     0;
      T     "DB_OP".M1_V_CPT;
_003: NOP   0;
      A     L 0.0;
      A(;
      A     "26S6";
      AN    "T_ALM2";
      A     "MM2_CONTADOR_FIN";
      O(;
      L     "DB_OP".M2_P_CPT;
      L     0;
      ==I;
      );
      );
      A(;
      L     "DB_OP".M1_P_CPT;
      L     0;
      <>I;
      );
      A     "Datos Pieza - Rolos".PiezaPresente;
      FP    "AuxFlanco2";
      JNB   _004;
      L     0;
      T     "DB_OP".M2_V_CPT;
_004: NOP   0;
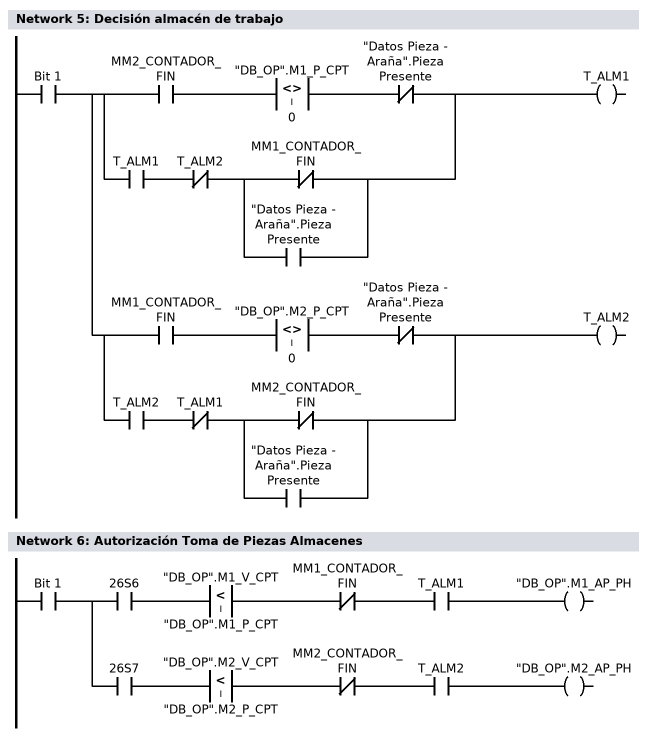
NETWORK
TITLE = Decisión almacén de trabajo
      A     "Bit 1";
      =     L 0.0;
      A     L 0.0;
      A(;
      A     "MM2_CONTADOR_FIN";
      A(;
      L     "DB_OP".M1_P_CPT;
      L     0;
      <>I;
      );
      AN    "Datos Pieza - Araña".PiezaPresente;
      O;
      A     "T_ALM1";
      AN    "T_ALM2";
      A(;
      ON    "MM1_CONTADOR_FIN";
      O     "Datos Pieza - Araña".PiezaPresente;
      );
      );
      =     "T_ALM1";
      A     L 0.0;
      A(;
      A     "MM1_CONTADOR_FIN";
      A(;
      L     "DB_OP".M2_P_CPT;
      L     0;
      <>I;
      );
      AN    "Datos Pieza - Araña".PiezaPresente;
      O;
      A     "T_ALM2";
      AN    "T_ALM1";
      A(;
      ON    "MM2_CONTADOR_FIN";
      O     "Datos Pieza - Araña".PiezaPresente;
      );
      );
      =     "T_ALM2";
NETWORK
TITLE = Autorización Toma de Piezas Almacenes
      A     "Bit 1";
      =     L 0.0;
      A     L 0.0;
      A     "26S6";
      A(;
      L     "DB_OP".M1_V_CPT;
      L     "DB_OP".M1_P_CPT;
      <I;
      );
      AN    "MM1_CONTADOR_FIN";
      A     "T_ALM1";
      =     "DB_OP".M1_AP_PH;
      A     L 0.0;
      A     "26S7";
      A(;
      L     "DB_OP".M2_V_CPT;
      L     "DB_OP".M2_P_CPT;
      <I;
      );
      AN    "MM2_CONTADOR_FIN";
      A     "T_ALM2";
      =     "DB_OP".M2_AP_PH;
END_FUNCTION

FUNCTION "Manual Selección Mov." : VOID	// FC 4
TITLE = Gestiona la selección de los movimientos manuales
VERSION : 0.1
VAR_TEMP
  Nmvt : WORD ;
END_VAR
BEGIN
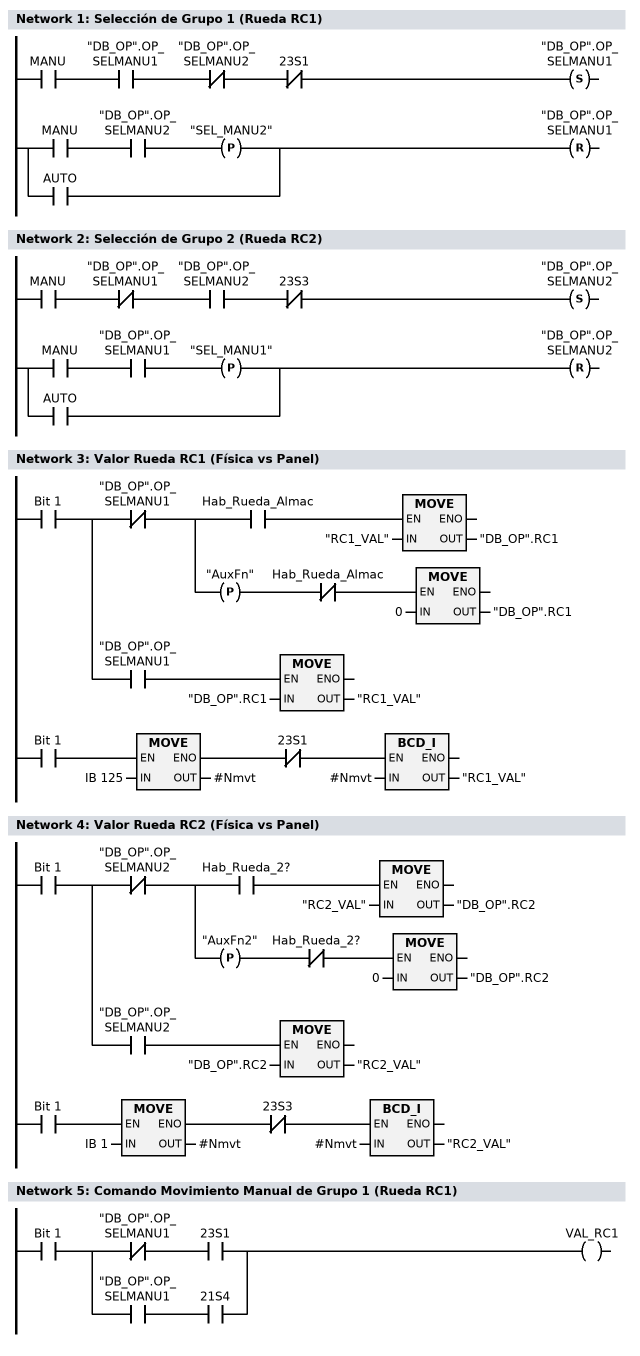
NETWORK
TITLE = Selección de Grupo 1 (Rueda RC1)
      A     "MANU";
      A     "DB_OP".OP_SELMANU1;
      AN    "DB_OP".OP_SELMANU2;
      AN    "23S1";
      S     "DB_OP".OP_SELMANU1;
      A(;
      A     "MANU";
      A     "DB_OP".OP_SELMANU2;
      FP    "SEL_MANU2";
      O     "AUTO";
      );
      R     "DB_OP".OP_SELMANU1;
      NOP   0;
NETWORK
TITLE = Selección de Grupo 2 (Rueda RC2)
      A     "MANU";
      AN    "DB_OP".OP_SELMANU1;
      A     "DB_OP".OP_SELMANU2;
      AN    "23S3";
      S     "DB_OP".OP_SELMANU2;
      A(;
      A     "MANU";
      A     "DB_OP".OP_SELMANU1;
      FP    "SEL_MANU1";
      O     "AUTO";
      );
      R     "DB_OP".OP_SELMANU2;
      NOP   0;
NETWORK
TITLE = Valor Rueda RC1 (Física vs Panel)
      A     "Bit 1";
      =     L 2.0;
      A(;
      A     L 2.0;
      JNB   _001;
      L     IB 125;
      T     #Nmvt;
      SET;
      SAVE;
      CLR;
_001: A     BR;
      );
      AN    "23S1";
      JNB   _002;
      L     #Nmvt;
      BTI;
      T     "RC1_VAL";
_002: NOP   0;
      A     L 2.0;
      AN    "DB_OP".OP_SELMANU1;
      =     L 2.1;
      A     L 2.1;
      A     "Hab_Rueda_Almac";
      JNB   _003;
      L     "RC1_VAL";
      T     "DB_OP".RC1;
_003: NOP   0;
      A     L 2.1;
      FP    "AuxFn";
      AN    "Hab_Rueda_Almac";
      JNB   _004;
      L     0;
      T     "DB_OP".RC1;
_004: NOP   0;
      A     L 2.0;
      A     "DB_OP".OP_SELMANU1;
      JNB   _005;
      L     "DB_OP".RC1;
      T     "RC1_VAL";
_005: NOP   0;
NETWORK
TITLE = Valor Rueda RC2 (Física vs Panel)
      A     "Bit 1";
      =     L 2.0;
      A(;
      A     L 2.0;
      JNB   _006;
      L     IB 1;
      T     #Nmvt;
      SET;
      SAVE;
      CLR;
_006: A     BR;
      );
      AN    "23S3";
      JNB   _007;
      L     #Nmvt;
      BTI;
      T     "RC2_VAL";
_007: NOP   0;
      A     L 2.0;
      AN    "DB_OP".OP_SELMANU2;
      =     L 2.1;
      A     L 2.1;
      A     "Hab_Rueda_2?";
      JNB   _008;
      L     "RC2_VAL";
      T     "DB_OP".RC2;
_008: NOP   0;
      A     L 2.1;
      FP    "AuxFn2";
      AN    "Hab_Rueda_2?";
      JNB   _009;
      L     0;
      T     "DB_OP".RC2;
_009: NOP   0;
      A     L 2.0;
      A     "DB_OP".OP_SELMANU2;
      JNB   _00a;
      L     "DB_OP".RC2;
      T     "RC2_VAL";
_00a: NOP   0;
NETWORK
TITLE = Comando Movimiento Manual de Grupo 1 (Rueda RC1)
      A     "Bit 1";
      A(;
      AN    "DB_OP".OP_SELMANU1;
      A     "23S1";
      O;
      A     "DB_OP".OP_SELMANU1;
      A     "21S4";
      );
      =     "VAL_RC1";
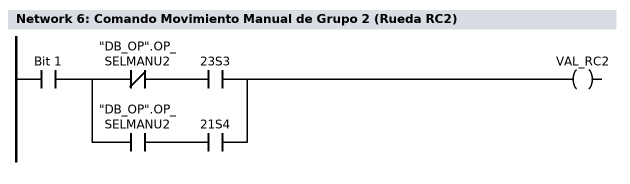
NETWORK
TITLE = Comando Movimiento Manual de Grupo 2 (Rueda RC2)
      A     "Bit 1";
      A(;
      AN    "DB_OP".OP_SELMANU2;
      A     "23S3";
      O;
      A     "DB_OP".OP_SELMANU2;
      A     "21S4";
      );
      =     "VAL_RC2";
END_FUNCTION

FUNCTION "General" : VOID	// FC 5
VERSION : 0.1
BEGIN
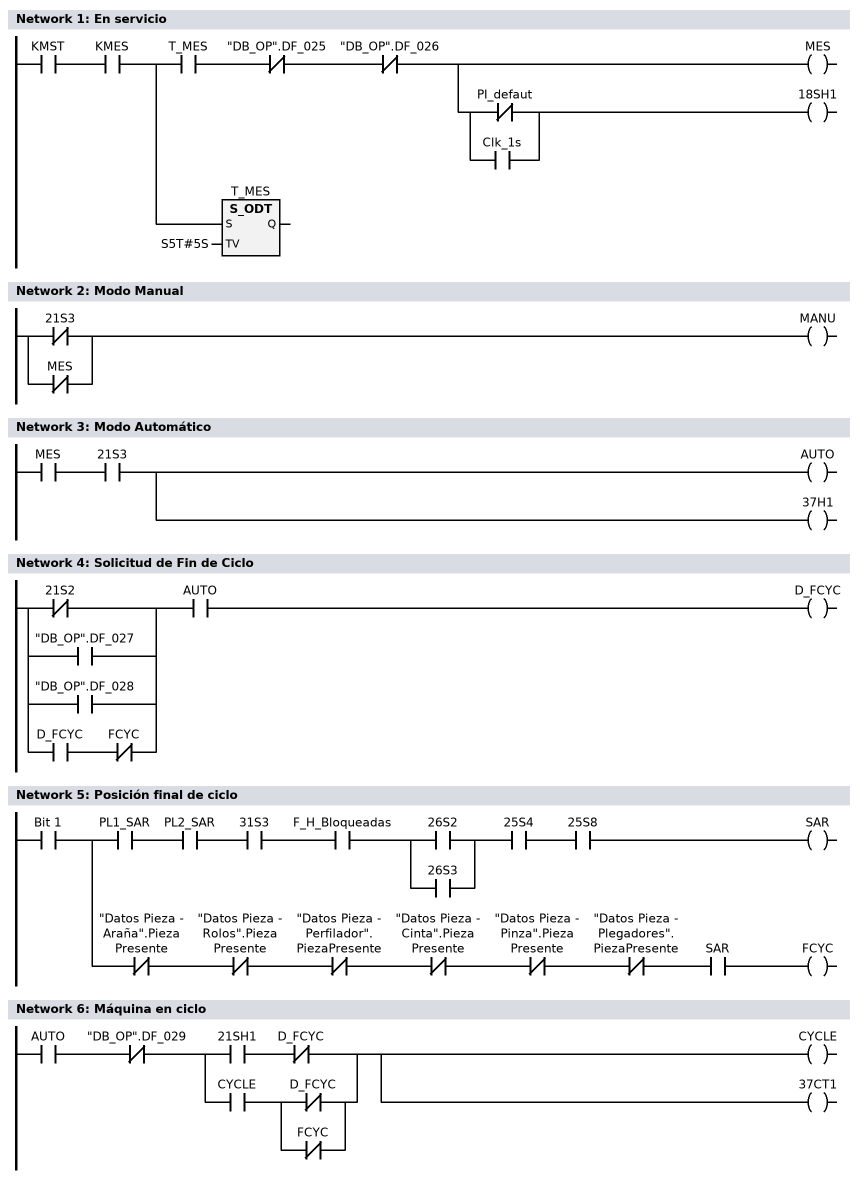
NETWORK
TITLE = En servicio
      A     "KMST";
      A     "KMES";
      =     L 0.0;
      A     L 0.0;
      A     "T_MES";
      AN    "DB_OP".DF_025;
      AN    "DB_OP".DF_026;
      =     L 0.1;
      A     L 0.1;
      BLD   102;
      =     "MES";
      A     L 0.1;
      A(;
      ON    "PI_defaut";
      O     "Clk_1s";
      );
      =     "18SH1";
      A     L 0.0;
      L     S5T#5S;
      SD    "T_MES";
      NOP   0;
      NOP   0;
      NOP   0;
      NOP   0;
NETWORK
TITLE = Modo Manual
      ON    "21S3";
      ON    "MES";
      =     "MANU";
NETWORK
TITLE = Modo Automático
      A     "MES";
      A     "21S3";
      =     "AUTO";
      =     "37H1";
NETWORK
TITLE = Solicitud de Fin de Ciclo
      A(;
      ON    "21S2";
      O     "DB_OP".DF_027;
      O     "DB_OP".DF_028;
      O;
      A     "D_FCYC";
      AN    "FCYC";
      );
      A     "AUTO";
      =     "D_FCYC";
NETWORK
TITLE = Posición final de ciclo
      A     "Bit 1";
      =     L 0.0;
      A     L 0.0;
      A     "PL1_SAR";
      A     "PL2_SAR";
      A     "31S3";
      A     "F_H_Bloqueadas";
      A(;
      O     "26S2";
      O     "26S3";
      );
      A     "25S4";
      A     "25S8";
      =     "SAR";
      A     L 0.0;
      AN    "Datos Pieza - Araña".PiezaPresente;
      AN    "Datos Pieza - Rolos".PiezaPresente;
      AN    "Datos Pieza - Perfilador".PiezaPresente;
      AN    "Datos Pieza - Cinta".PiezaPresente;
      AN    "Datos Pieza - Pinza".PiezaPresente;
      AN    "Datos Pieza - Plegadores".PiezaPresente;
      A     "SAR";
      =     "FCYC";
NETWORK
TITLE = Máquina en ciclo
      A     "AUTO";
      AN    "DB_OP".DF_029;
      A(;
      A     "21SH1";
      AN    "D_FCYC";
      O;
      A     "CYCLE";
      A(;
      ON    "D_FCYC";
      ON    "FCYC";
      );
      );
      =     "CYCLE";
      =     "37CT1";
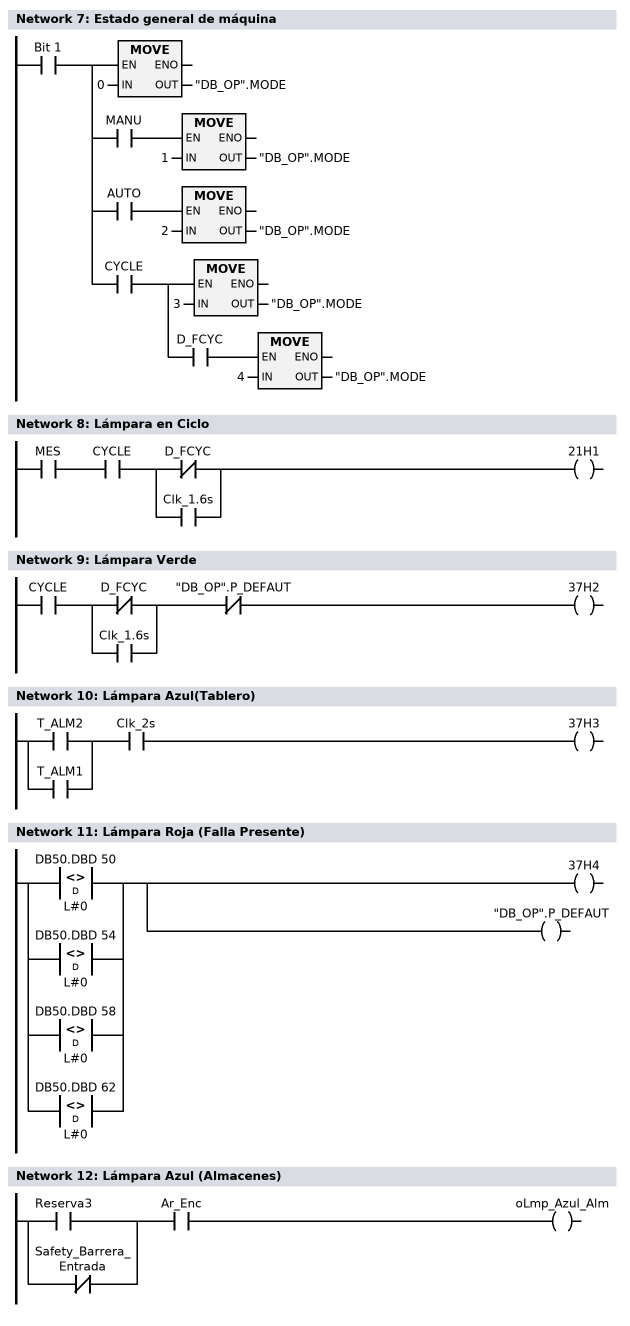
NETWORK
TITLE = Estado general de máquina
      A     "Bit 1";
      =     L 0.0;
      A     L 0.0;
      JNB   _001;
      L     0;
      T     "DB_OP".MODE;
_001: NOP   0;
      A     L 0.0;
      A     "MANU";
      JNB   _002;
      L     1;
      T     "DB_OP".MODE;
_002: NOP   0;
      A     L 0.0;
      A     "AUTO";
      JNB   _003;
      L     2;
      T     "DB_OP".MODE;
_003: NOP   0;
      A     L 0.0;
      A     "CYCLE";
      =     L 0.1;
      A     L 0.1;
      JNB   _004;
      L     3;
      T     "DB_OP".MODE;
_004: NOP   0;
      A     L 0.1;
      A     "D_FCYC";
      JNB   _005;
      L     4;
      T     "DB_OP".MODE;
_005: NOP   0;
NETWORK
TITLE = Lámpara en Ciclo
      A     "MES";
      A     "CYCLE";
      A(;
      ON    "D_FCYC";
      O     "Clk_1.6s";
      );
      =     "21H1";
NETWORK
TITLE = Lámpara Verde
      A     "CYCLE";
      A(;
      ON    "D_FCYC";
      O     "Clk_1.6s";
      );
      AN    "DB_OP".P_DEFAUT;
      =     "37H2";
NETWORK
TITLE = Lámpara Azul(Tablero)
      A(;
      O     "T_ALM2";
      O     "T_ALM1";
      );
      A     "Clk_2s";
      =     "37H3";
NETWORK
TITLE = Lámpara Roja (Falla Presente)
      O(;
      L     DB50.DBD 50;
      L     L#0;
      <>D;
      );
      O(;
      L     DB50.DBD 54;
      L     L#0;
      <>D;
      );
      O(;
      L     DB50.DBD 58;
      L     L#0;
      <>D;
      );
      O(;
      L     DB50.DBD 62;
      L     L#0;
      <>D;
      );
      =     "37H4";
      =     "DB_OP".P_DEFAUT;
NETWORK
TITLE = Lámpara Azul (Almacenes)
      A(;
      O     "Reserva3";
      ON    "Safety_Barrera_Entrada";
      );
      A     "Ar_Enc";
      =     "oLmp_Azul_Alm";
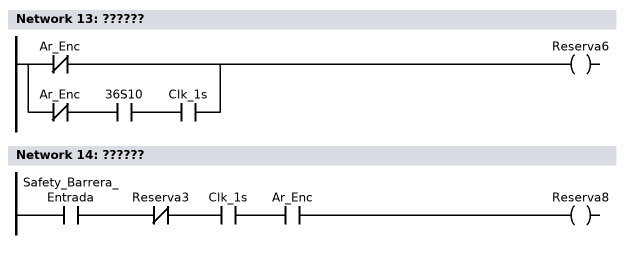
NETWORK
TITLE = ??????
      ON    "Ar_Enc";
      O;
      AN    "Ar_Enc";
      A     "36S10";
      A     "Clk_1s";
      =     "Reserva6";
NETWORK
TITLE = ??????
      A     "Safety_Barrera_Entrada";
      AN    "Reserva3";
      A     "Clk_1s";
      A     "Ar_Enc";
      =     "Reserva8";
END_FUNCTION

